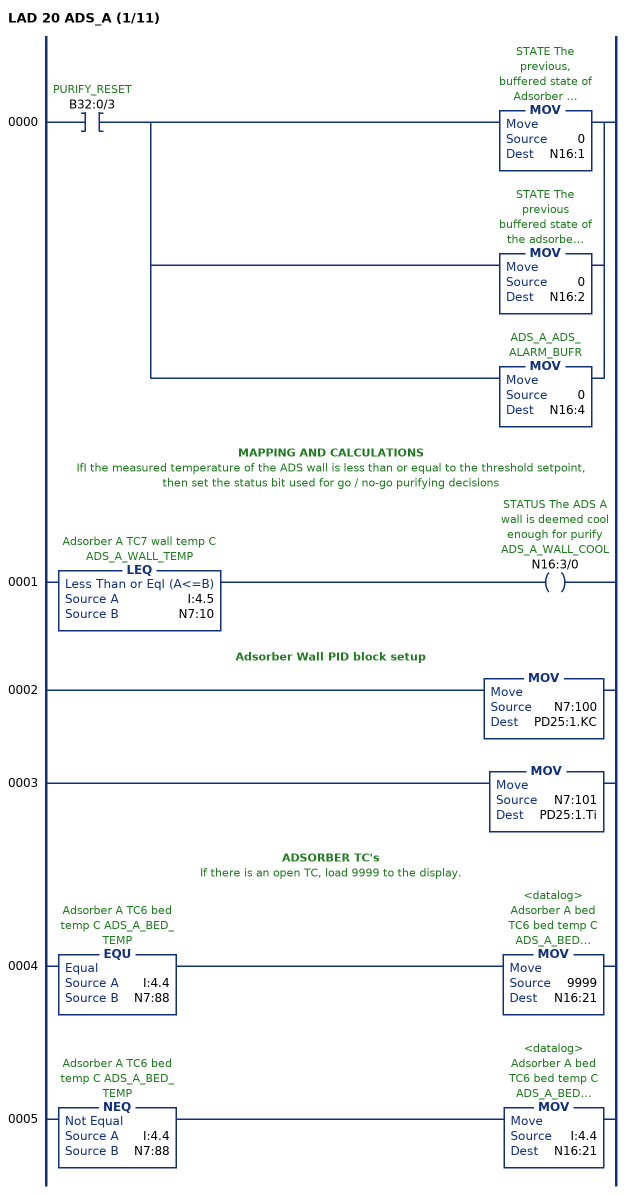
% Rung: 0 %
SOR XIC B32:0/3 BST MOV 0 N16:1 NXB MOV 0 N16:2 NXB MOV 0 N16:4 BND EOR
%   B32:0/3  PURIFY_RESET %
%   N16:1  ADS_A_STANDBY_BUFFER  "STATE The previous, buffered state of Adsorber A" %
%   N16:2  ADS_A_SYS_ALARM_BUFR  "STATE The previous buffered state of the adsorber when the alarm occured" %
%   N16:4  ADS_A_ADS_ALARM_BUFR %
% Rung: 1 %
% TITLE: MAPPING AND CALCULATIONS %
% IfI the measured temperature of the ADS wall is less than or equal to the threshold setpoint, then set the status bit used for go / no-go purifying decisions %
SOR LEQ I:4.5 N7:10 OTE N16:3/0 EOR
%   I:4.5  ADS_A_WALL_TEMP  "Adsorber A TC7 wall temp C" %
%   N7:10  ADS_WALL_TEMP_COOL  "CONFIG The temp at which the adsorber wall is deemed to be cool enough to purify" %
%   N16:3/0  ADS_A_WALL_COOL  "STATUS The ADS A wall is deemed cool enough for purify" %
% Rung: 2 %
% TITLE: Adsorber Wall PID block setup %
SOR MOV N7:100 PD25:1.KC EOR
%   N7:100  BLANKET_P  "CONFIG Blanket Proportional Gain New" %
% Rung: 3 %
SOR MOV N7:101 PD25:1.Ti EOR
%   N7:101  BLANKET_I  "CONFIG Blanket Integral Gain New" %
% Rung: 4 %
% TITLE: ADSORBER TC's %
% If there is an open TC, load 9999 to the display. %
SOR EQU I:4.4 N7:88 MOV 9999 N16:21 EOR
%   I:4.4  ADS_A_BED_TEMP  "Adsorber A TC6 bed temp C" %
%   N7:88  TC_OPEN_SP  "CONFIG The value read by an open TC input" %
%   N16:21  ADS_A_BED_TEMP_READ  "<datalog> Adsorber A bed TC6 bed temp C" %
% Rung: 5 %
SOR NEQ I:4.4 N7:88 MOV I:4.4 N16:21 EOR
%   I:4.4  ADS_A_BED_TEMP  "Adsorber A TC6 bed temp C" %
%   N7:88  TC_OPEN_SP  "CONFIG The value read by an open TC input" %
%   N16:21  ADS_A_BED_TEMP_READ  "<datalog> Adsorber A bed TC6 bed temp C" %

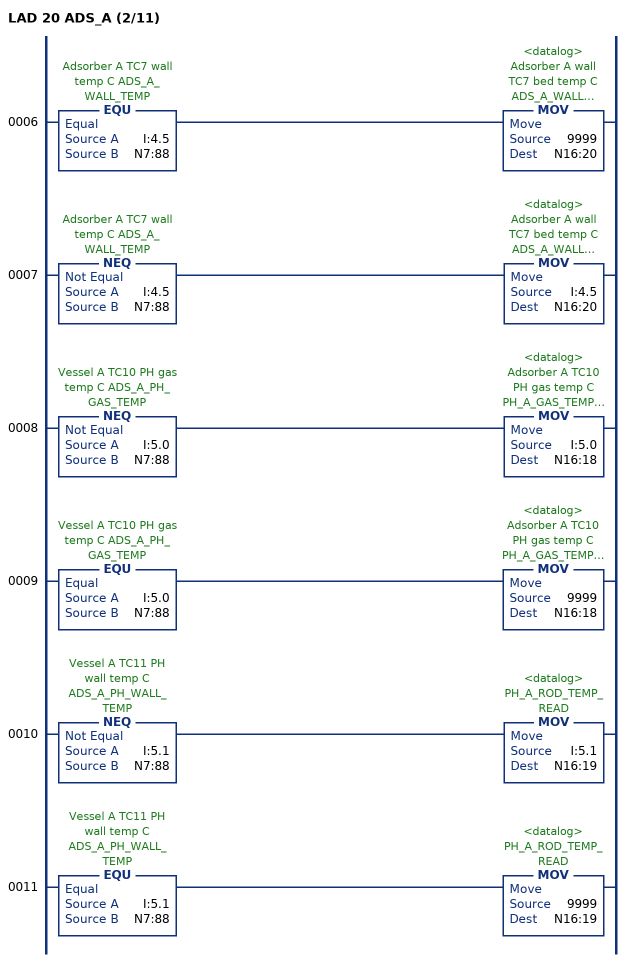
% Rung: 6 %
SOR EQU I:4.5 N7:88 MOV 9999 N16:20 EOR
%   I:4.5  ADS_A_WALL_TEMP  "Adsorber A TC7 wall temp C" %
%   N7:88  TC_OPEN_SP  "CONFIG The value read by an open TC input" %
%   N16:20  ADS_A_WALL_TEMP_READ  "<datalog> Adsorber A wall TC7 bed temp C" %
% Rung: 7 %
SOR NEQ I:4.5 N7:88 MOV I:4.5 N16:20 EOR
%   I:4.5  ADS_A_WALL_TEMP  "Adsorber A TC7 wall temp C" %
%   N7:88  TC_OPEN_SP  "CONFIG The value read by an open TC input" %
%   N16:20  ADS_A_WALL_TEMP_READ  "<datalog> Adsorber A wall TC7 bed temp C" %
% Rung: 8 %
SOR NEQ I:5.0 N7:88 MOV I:5.0 N16:18 EOR
%   I:5.0  ADS_A_PH_GAS_TEMP  "Vessel A TC10 PH gas temp C" %
%   N7:88  TC_OPEN_SP  "CONFIG The value read by an open TC input" %
%   N16:18  PH_A_GAS_TEMP_READ  "<datalog> Adsorber A TC10 PH gas temp C" %
% Rung: 9 %
SOR EQU I:5.0 N7:88 MOV 9999 N16:18 EOR
%   I:5.0  ADS_A_PH_GAS_TEMP  "Vessel A TC10 PH gas temp C" %
%   N7:88  TC_OPEN_SP  "CONFIG The value read by an open TC input" %
%   N16:18  PH_A_GAS_TEMP_READ  "<datalog> Adsorber A TC10 PH gas temp C" %
% Rung: 10 %
SOR NEQ I:5.1 N7:88 MOV I:5.1 N16:19 EOR
%   I:5.1  ADS_A_PH_WALL_TEMP  "Vessel A TC11 PH wall temp C" %
%   N7:88  TC_OPEN_SP  "CONFIG The value read by an open TC input" %
%   N16:19  PH_A_ROD_TEMP_READ  "<datalog>" %
% Rung: 11 %
SOR EQU I:5.1 N7:88 MOV 9999 N16:19 EOR
%   I:5.1  ADS_A_PH_WALL_TEMP  "Vessel A TC11 PH wall temp C" %
%   N7:88  TC_OPEN_SP  "CONFIG The value read by an open TC input" %
%   N16:19  PH_A_ROD_TEMP_READ  "<datalog>" %

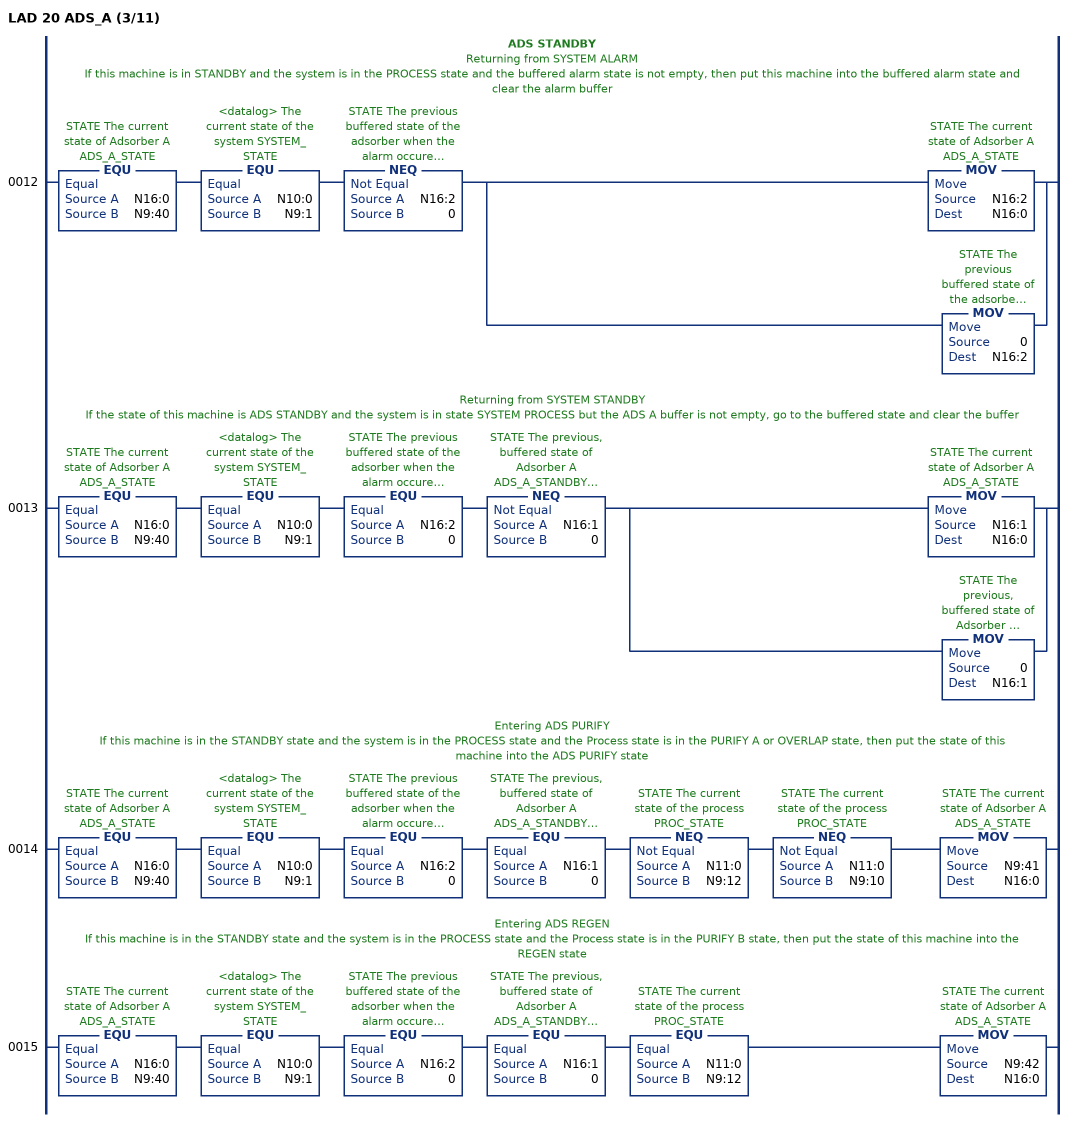
% Rung: 12 %
% TITLE: ADS STANDBY %
% Returning from SYSTEM ALARM
% If this machine is in STANDBY and the system is in the PROCESS state and the buffered alarm state is not empty, then put this machine into the buffered alarm state and clear the alarm buffer %
SOR EQU N16:0 N9:40 EQU N10:0 N9:1 NEQ N16:2 0 BST MOV N16:2 N16:0 NXB MOV 0 N16:2 BND EOR
%   N16:0  ADS_A_STATE  "STATE The current state of Adsorber A" %
%   N9:40  ADS_STANDBY  "STATE ADS Standby" %
%   N10:0  SYSTEM_STATE  "<datalog> The current state of the system" %
%   N9:1  SYSTEM_PROCESS  "STATE System Process" %
%   N16:2  ADS_A_SYS_ALARM_BUFR  "STATE The previous buffered state of the adsorber when the alarm occured" %
% Rung: 13 %
% Returning from SYSTEM STANDBY
% If the state of this machine is ADS STANDBY and the system is in state SYSTEM PROCESS but the ADS A buffer is not empty, go to the buffered state and clear the buffer %
SOR EQU N16:0 N9:40 EQU N10:0 N9:1 EQU N16:2 0 NEQ N16:1 0 BST MOV N16:1 N16:0 NXB MOV 0 N16:1 BND EOR
%   N16:0  ADS_A_STATE  "STATE The current state of Adsorber A" %
%   N9:40  ADS_STANDBY  "STATE ADS Standby" %
%   N10:0  SYSTEM_STATE  "<datalog> The current state of the system" %
%   N9:1  SYSTEM_PROCESS  "STATE System Process" %
%   N16:2  ADS_A_SYS_ALARM_BUFR  "STATE The previous buffered state of the adsorber when the alarm occured" %
%   N16:1  ADS_A_STANDBY_BUFFER  "STATE The previous, buffered state of Adsorber A" %
% Rung: 14 %
% Entering ADS PURIFY
% If this machine is in the STANDBY state and the system is in the PROCESS state and the Process state is in the PURIFY A or OVERLAP state, then put the state of this machine into the ADS PURIFY state %
SOR EQU N16:0 N9:40 EQU N10:0 N9:1 EQU N16:2 0 EQU N16:1 0 NEQ N11:0 N9:12 NEQ N11:0 N9:10 MOV N9:41 N16:0 EOR
%   N16:0  ADS_A_STATE  "STATE The current state of Adsorber A" %
%   N9:40  ADS_STANDBY  "STATE ADS Standby" %
%   N10:0  SYSTEM_STATE  "<datalog> The current state of the system" %
%   N9:1  SYSTEM_PROCESS  "STATE System Process" %
%   N16:2  ADS_A_SYS_ALARM_BUFR  "STATE The previous buffered state of the adsorber when the alarm occured" %
%   N16:1  ADS_A_STANDBY_BUFFER  "STATE The previous, buffered state of Adsorber A" %
%   N11:0  PROC_STATE  "STATE The current state of the process" %
%   N9:12  PROC_REGEN_A  "STATE Process Purify B" %
%   N9:10  PROCESS_STANDBY %
%   N9:41  ADS_PURIFY  "STATE ADS Purify" %
% Rung: 15 %
% Entering ADS REGEN
% If this machine is in the STANDBY state and the system is in the PROCESS state and the Process state is in the PURIFY B state, then put the state of this machine into the REGEN state %
SOR EQU N16:0 N9:40 EQU N10:0 N9:1 EQU N16:2 0 EQU N16:1 0 EQU N11:0 N9:12 MOV N9:42 N16:0 EOR
%   N16:0  ADS_A_STATE  "STATE The current state of Adsorber A" %
%   N9:40  ADS_STANDBY  "STATE ADS Standby" %
%   N10:0  SYSTEM_STATE  "<datalog> The current state of the system" %
%   N9:1  SYSTEM_PROCESS  "STATE System Process" %
%   N16:2  ADS_A_SYS_ALARM_BUFR  "STATE The previous buffered state of the adsorber when the alarm occured" %
%   N16:1  ADS_A_STANDBY_BUFFER  "STATE The previous, buffered state of Adsorber A" %
%   N11:0  PROC_STATE  "STATE The current state of the process" %
%   N9:12  PROC_REGEN_A  "STATE Process Purify B" %
%   N9:42  ADS_REGEN  "STATE ADS Regen" %

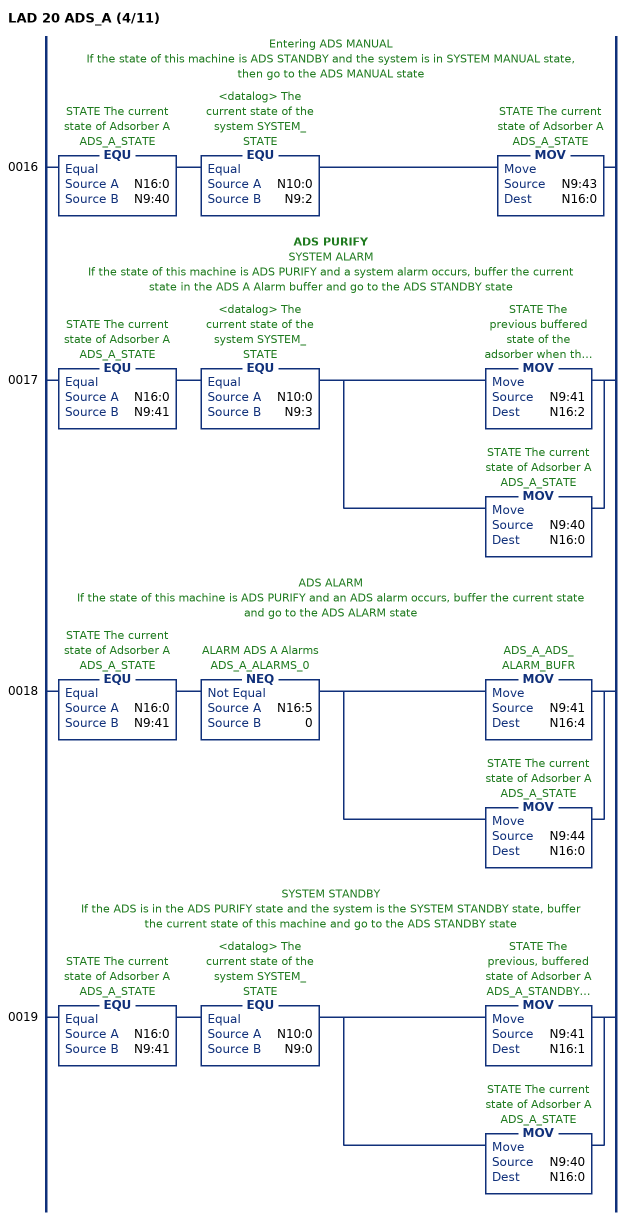
% Rung: 16 %
% Entering ADS MANUAL
% If the state of this machine is ADS STANDBY and the system is in SYSTEM MANUAL state, then go to the ADS MANUAL state %
SOR EQU N16:0 N9:40 EQU N10:0 N9:2 MOV N9:43 N16:0 EOR
%   N16:0  ADS_A_STATE  "STATE The current state of Adsorber A" %
%   N9:40  ADS_STANDBY  "STATE ADS Standby" %
%   N10:0  SYSTEM_STATE  "<datalog> The current state of the system" %
%   N9:2  SYSTEM_MANUAL  "STATE System Manual" %
%   N9:43  ADS_MANUAL  "STATE ADS Manual" %
% Rung: 17 %
% TITLE: ADS PURIFY %
% SYSTEM ALARM
% If the state of this machine is ADS PURIFY and a system alarm occurs, buffer the current state in the ADS A Alarm buffer and go to the ADS STANDBY state %
SOR EQU N16:0 N9:41 EQU N10:0 N9:3 BST MOV N9:41 N16:2 NXB MOV N9:40 N16:0 BND EOR
%   N16:0  ADS_A_STATE  "STATE The current state of Adsorber A" %
%   N9:41  ADS_PURIFY  "STATE ADS Purify" %
%   N10:0  SYSTEM_STATE  "<datalog> The current state of the system" %
%   N9:3  SYSTEM_ALARM  "STATE System Alarm" %
%   N16:2  ADS_A_SYS_ALARM_BUFR  "STATE The previous buffered state of the adsorber when the alarm occured" %
%   N9:40  ADS_STANDBY  "STATE ADS Standby" %
% Rung: 18 %
% ADS ALARM
% If the state of this machine is ADS PURIFY and an ADS alarm occurs, buffer the current state and go to the ADS ALARM state %
SOR EQU N16:0 N9:41 NEQ N16:5 0 BST MOV N9:41 N16:4 NXB MOV N9:44 N16:0 BND EOR
%   N16:0  ADS_A_STATE  "STATE The current state of Adsorber A" %
%   N9:41  ADS_PURIFY  "STATE ADS Purify" %
%   N16:5  ADS_A_ALARMS_0  "ALARM ADS A Alarms" %
%   N16:4  ADS_A_ADS_ALARM_BUFR %
%   N9:44  ADS_ALARM  "STATE ADS Alarm" %
% Rung: 19 %
% SYSTEM STANDBY
% If the ADS is in the ADS PURIFY state and the system is the SYSTEM STANDBY state, buffer the current state of this machine and go to the ADS STANDBY state %
SOR EQU N16:0 N9:41 EQU N10:0 N9:0 BST MOV N9:41 N16:1 NXB MOV N9:40 N16:0 BND EOR
%   N16:0  ADS_A_STATE  "STATE The current state of Adsorber A" %
%   N9:41  ADS_PURIFY  "STATE ADS Purify" %
%   N10:0  SYSTEM_STATE  "<datalog> The current state of the system" %
%   N9:0  SYSTEM_STANDBY  "STATE System Standby" %
%   N16:1  ADS_A_STANDBY_BUFFER  "STATE The previous, buffered state of Adsorber A" %
%   N9:40  ADS_STANDBY  "STATE ADS Standby" %

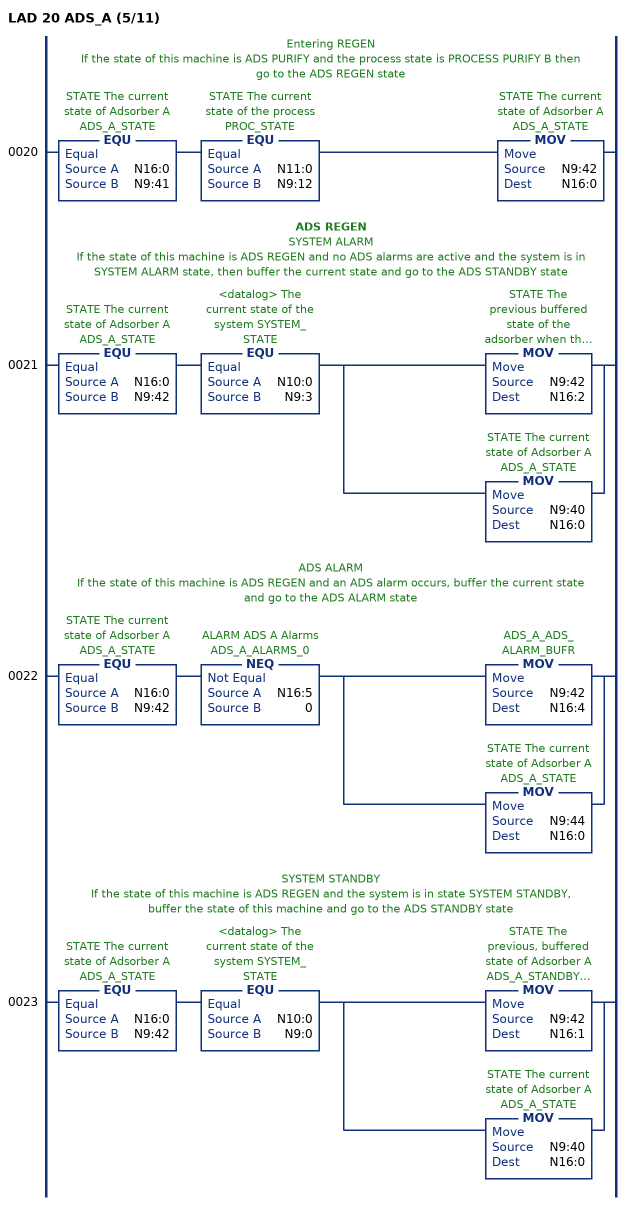
% Rung: 20 %
% Entering REGEN
% If the state of this machine is ADS PURIFY and the process state is PROCESS PURIFY B then go to the ADS REGEN state %
SOR EQU N16:0 N9:41 EQU N11:0 N9:12 MOV N9:42 N16:0 EOR
%   N16:0  ADS_A_STATE  "STATE The current state of Adsorber A" %
%   N9:41  ADS_PURIFY  "STATE ADS Purify" %
%   N11:0  PROC_STATE  "STATE The current state of the process" %
%   N9:12  PROC_REGEN_A  "STATE Process Purify B" %
%   N9:42  ADS_REGEN  "STATE ADS Regen" %
% Rung: 21 %
% TITLE: ADS REGEN %
% SYSTEM ALARM
% If the state of this machine is ADS REGEN and no ADS alarms are active and the system is in SYSTEM ALARM state, then buffer the current state and go to the ADS STANDBY state %
SOR EQU N16:0 N9:42 EQU N10:0 N9:3 BST MOV N9:42 N16:2 NXB MOV N9:40 N16:0 BND EOR
%   N16:0  ADS_A_STATE  "STATE The current state of Adsorber A" %
%   N9:42  ADS_REGEN  "STATE ADS Regen" %
%   N10:0  SYSTEM_STATE  "<datalog> The current state of the system" %
%   N9:3  SYSTEM_ALARM  "STATE System Alarm" %
%   N16:2  ADS_A_SYS_ALARM_BUFR  "STATE The previous buffered state of the adsorber when the alarm occured" %
%   N9:40  ADS_STANDBY  "STATE ADS Standby" %
% Rung: 22 %
% ADS ALARM
% If the state of this machine is ADS REGEN and an ADS alarm occurs, buffer the current state and go to the ADS ALARM state %
SOR EQU N16:0 N9:42 NEQ N16:5 0 BST MOV N9:42 N16:4 NXB MOV N9:44 N16:0 BND EOR
%   N16:0  ADS_A_STATE  "STATE The current state of Adsorber A" %
%   N9:42  ADS_REGEN  "STATE ADS Regen" %
%   N16:5  ADS_A_ALARMS_0  "ALARM ADS A Alarms" %
%   N16:4  ADS_A_ADS_ALARM_BUFR %
%   N9:44  ADS_ALARM  "STATE ADS Alarm" %
% Rung: 23 %
% SYSTEM STANDBY
% If the state of this machine is ADS REGEN and the system is in state SYSTEM STANDBY, buffer the state of this machine and go to the ADS STANDBY state %
SOR EQU N16:0 N9:42 EQU N10:0 N9:0 BST MOV N9:42 N16:1 NXB MOV N9:40 N16:0 BND EOR
%   N16:0  ADS_A_STATE  "STATE The current state of Adsorber A" %
%   N9:42  ADS_REGEN  "STATE ADS Regen" %
%   N10:0  SYSTEM_STATE  "<datalog> The current state of the system" %
%   N9:0  SYSTEM_STANDBY  "STATE System Standby" %
%   N16:1  ADS_A_STANDBY_BUFFER  "STATE The previous, buffered state of Adsorber A" %
%   N9:40  ADS_STANDBY  "STATE ADS Standby" %

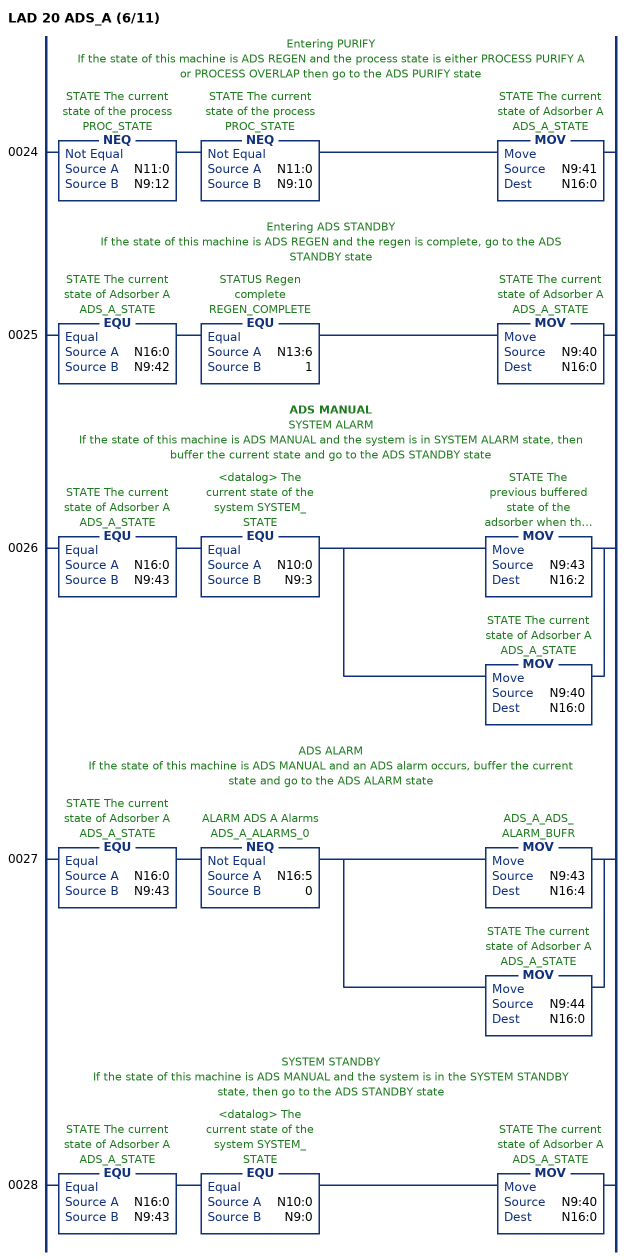
% Rung: 24 %
% Entering PURIFY
% If the state of this machine is ADS REGEN and the process state is either PROCESS PURIFY A or PROCESS OVERLAP then go to the ADS PURIFY state %
SOR NEQ N11:0 N9:12 NEQ N11:0 N9:10 MOV N9:41 N16:0 EOR
%   N11:0  PROC_STATE  "STATE The current state of the process" %
%   N9:12  PROC_REGEN_A  "STATE Process Purify B" %
%   N9:10  PROCESS_STANDBY %
%   N9:41  ADS_PURIFY  "STATE ADS Purify" %
%   N16:0  ADS_A_STATE  "STATE The current state of Adsorber A" %
% Rung: 25 %
% Entering ADS STANDBY
% If the state of this machine is ADS REGEN and the regen is complete, go to the ADS STANDBY state %
SOR EQU N16:0 N9:42 EQU N13:6 1 MOV N9:40 N16:0 EOR
%   N16:0  ADS_A_STATE  "STATE The current state of Adsorber A" %
%   N9:42  ADS_REGEN  "STATE ADS Regen" %
%   N13:6  REGEN_COMPLETE  "STATUS Regen complete" %
%   N9:40  ADS_STANDBY  "STATE ADS Standby" %
% Rung: 26 %
% TITLE: ADS MANUAL %
% SYSTEM ALARM
% If the state of this machine is ADS MANUAL and the system is in SYSTEM ALARM state, then buffer the current state and go to the ADS STANDBY state %
SOR EQU N16:0 N9:43 EQU N10:0 N9:3 BST MOV N9:43 N16:2 NXB MOV N9:40 N16:0 BND EOR
%   N16:0  ADS_A_STATE  "STATE The current state of Adsorber A" %
%   N9:43  ADS_MANUAL  "STATE ADS Manual" %
%   N10:0  SYSTEM_STATE  "<datalog> The current state of the system" %
%   N9:3  SYSTEM_ALARM  "STATE System Alarm" %
%   N16:2  ADS_A_SYS_ALARM_BUFR  "STATE The previous buffered state of the adsorber when the alarm occured" %
%   N9:40  ADS_STANDBY  "STATE ADS Standby" %
% Rung: 27 %
% ADS ALARM
% If the state of this machine is ADS MANUAL and an ADS alarm occurs, buffer the current state and go to the ADS ALARM state %
SOR EQU N16:0 N9:43 NEQ N16:5 0 BST MOV N9:43 N16:4 NXB MOV N9:44 N16:0 BND EOR
%   N16:0  ADS_A_STATE  "STATE The current state of Adsorber A" %
%   N9:43  ADS_MANUAL  "STATE ADS Manual" %
%   N16:5  ADS_A_ALARMS_0  "ALARM ADS A Alarms" %
%   N16:4  ADS_A_ADS_ALARM_BUFR %
%   N9:44  ADS_ALARM  "STATE ADS Alarm" %
% Rung: 28 %
% SYSTEM STANDBY
% If the state of this machine is ADS MANUAL and the system is in the SYSTEM STANDBY state, then go to the ADS STANDBY state %
SOR EQU N16:0 N9:43 EQU N10:0 N9:0 MOV N9:40 N16:0 EOR
%   N16:0  ADS_A_STATE  "STATE The current state of Adsorber A" %
%   N9:43  ADS_MANUAL  "STATE ADS Manual" %
%   N10:0  SYSTEM_STATE  "<datalog> The current state of the system" %
%   N9:0  SYSTEM_STANDBY  "STATE System Standby" %
%   N9:40  ADS_STANDBY  "STATE ADS Standby" %

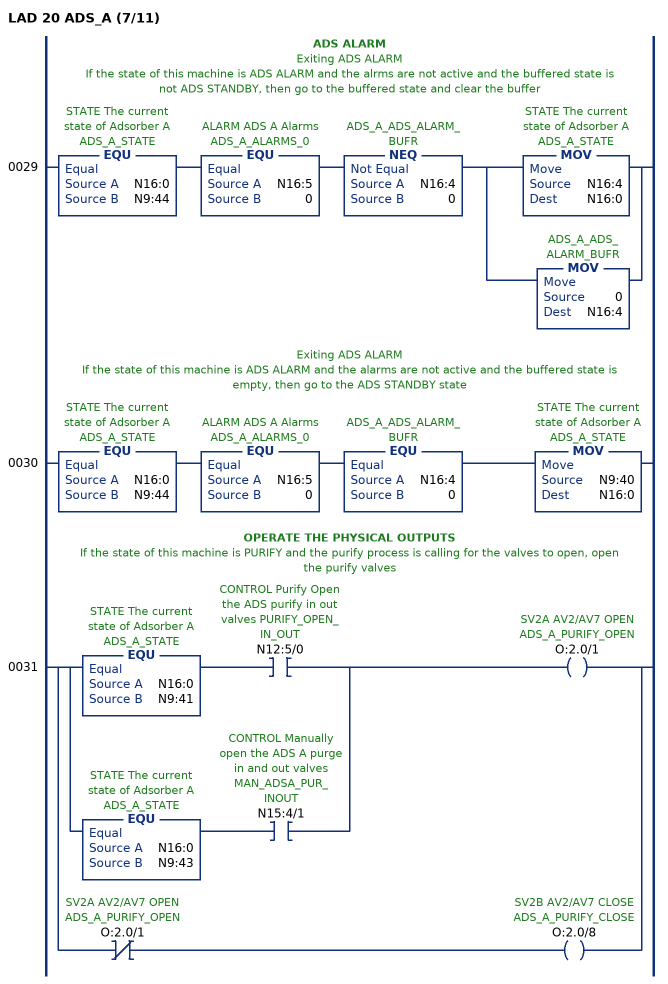
% Rung: 29 %
% TITLE: ADS ALARM %
% Exiting ADS ALARM
% If the state of this machine is ADS ALARM and the alrms are not active and the buffered state is not ADS STANDBY, then go to the buffered state and clear the buffer %
SOR EQU N16:0 N9:44 EQU N16:5 0 NEQ N16:4 0 BST MOV N16:4 N16:0 NXB MOV 0 N16:4 BND EOR
%   N16:0  ADS_A_STATE  "STATE The current state of Adsorber A" %
%   N9:44  ADS_ALARM  "STATE ADS Alarm" %
%   N16:5  ADS_A_ALARMS_0  "ALARM ADS A Alarms" %
%   N16:4  ADS_A_ADS_ALARM_BUFR %
% Rung: 30 %
% Exiting ADS ALARM
% If the state of this machine is ADS ALARM and the alarms are not active and the buffered state is empty, then go to the ADS STANDBY state %
SOR EQU N16:0 N9:44 EQU N16:5 0 EQU N16:4 0 MOV N9:40 N16:0 EOR
%   N16:0  ADS_A_STATE  "STATE The current state of Adsorber A" %
%   N9:44  ADS_ALARM  "STATE ADS Alarm" %
%   N16:5  ADS_A_ALARMS_0  "ALARM ADS A Alarms" %
%   N16:4  ADS_A_ADS_ALARM_BUFR %
%   N9:40  ADS_STANDBY  "STATE ADS Standby" %
% Rung: 31 %
% TITLE: OPERATE THE PHYSICAL OUTPUTS %
% If the state of this machine is PURIFY and the purify process is calling for the valves to open, open the purify valves %
SOR BST BST EQU N16:0 N9:41 XIC N12:5/0 NXB EQU N16:0 N9:43 XIC N15:4/1 BND OTE O:2.0/1 NXB XIO O:2.0/1 OTE O:2.0/8 BND EOR
%   N16:0  ADS_A_STATE  "STATE The current state of Adsorber A" %
%   N9:41  ADS_PURIFY  "STATE ADS Purify" %
%   N12:5/0  PURIFY_OPEN_IN_OUT  "CONTROL Purify Open the ADS purify in out valves" %
%   N9:43  ADS_MANUAL  "STATE ADS Manual" %
%   N15:4/1  MAN_ADSA_PUR_INOUT  "CONTROL Manually open the ADS A purge in and out valves" %
%   O:2.0/1  ADS_A_PURIFY_OPEN  "SV2A AV2/AV7 OPEN" %
%   O:2.0/8  ADS_A_PURIFY_CLOSE  "SV2B AV2/AV7 CLOSE" %

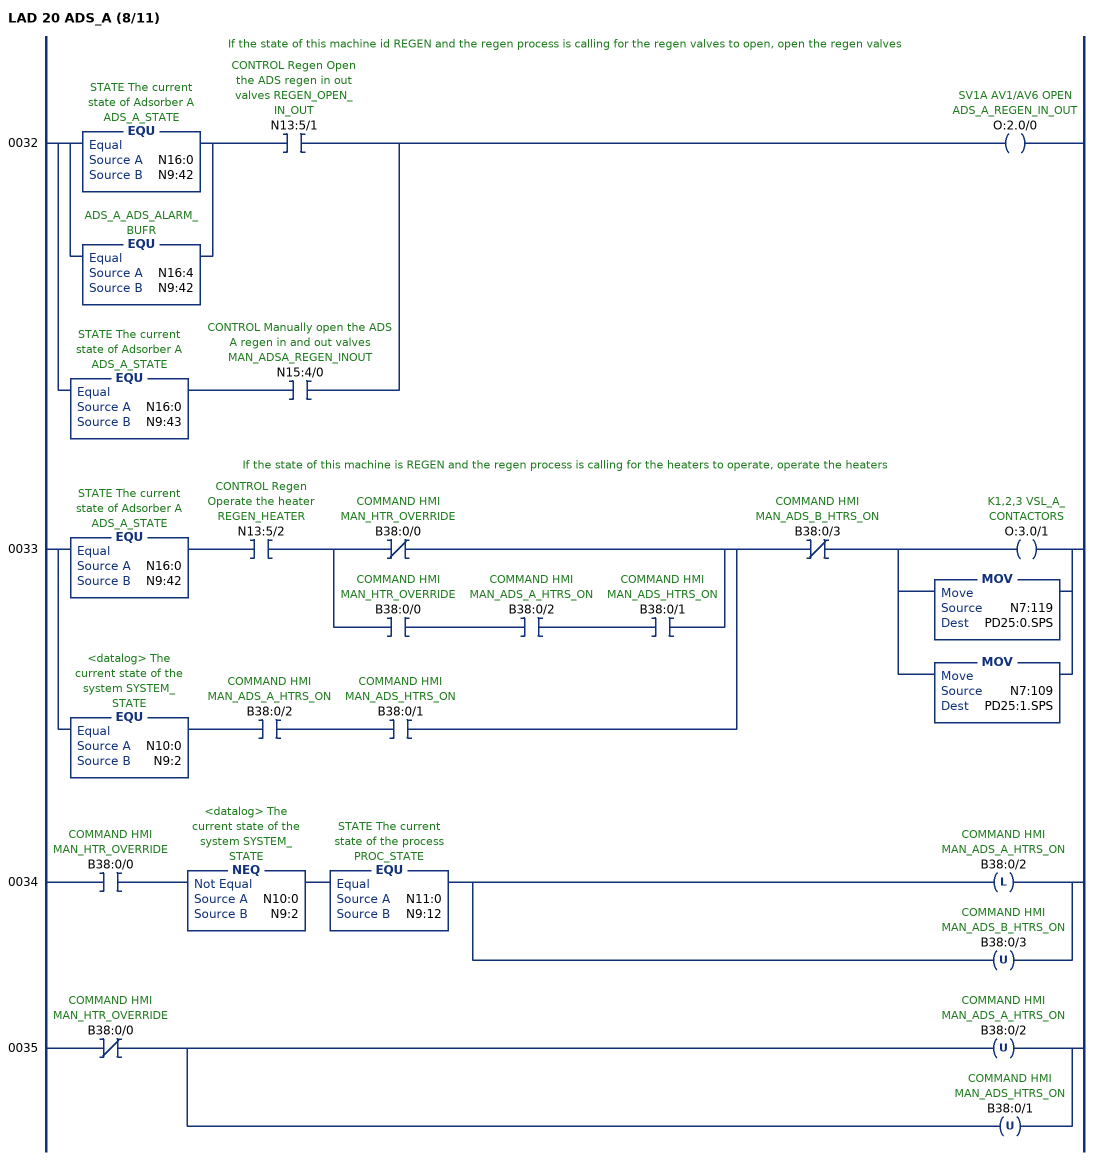
% Rung: 32 %
% If the state of this machine id REGEN and the regen process is calling for the regen valves to open, open the regen valves %
SOR BST BST EQU N16:0 N9:42 NXB EQU N16:4 N9:42 BND XIC N13:5/1 NXB EQU N16:0 N9:43 XIC N15:4/0 BND OTE O:2.0/0 EOR
%   N16:0  ADS_A_STATE  "STATE The current state of Adsorber A" %
%   N9:42  ADS_REGEN  "STATE ADS Regen" %
%   N16:4  ADS_A_ADS_ALARM_BUFR %
%   N13:5/1  REGEN_OPEN_IN_OUT  "CONTROL Regen Open the ADS regen in out valves" %
%   N9:43  ADS_MANUAL  "STATE ADS Manual" %
%   N15:4/0  MAN_ADSA_REGEN_INOUT  "CONTROL Manually open the ADS A regen in and out valves" %
%   O:2.0/0  ADS_A_REGEN_IN_OUT  "SV1A AV1/AV6 OPEN" %
% Rung: 33 %
% If the state of this machine is REGEN and the regen process is calling for the heaters to operate, operate the heaters %
SOR BST EQU N16:0 N9:42 XIC N13:5/2 BST XIO B38:0/0 NXB XIC B38:0/0 XIC B38:0/2 XIC B38:0/1 BND NXB EQU N10:0 N9:2 XIC B38:0/2 XIC B38:0/1 BND XIO B38:0/3 BST OTE O:3.0/1 NXB MOV N7:119 PD25:0.SPS NXB MOV N7:109 PD25:1.SPS BND EOR
%   N16:0  ADS_A_STATE  "STATE The current state of Adsorber A" %
%   N9:42  ADS_REGEN  "STATE ADS Regen" %
%   N13:5/2  REGEN_HEATER  "CONTROL Regen Operate the heater" %
%   B38:0/0  MAN_HTR_OVERRIDE  "COMMAND HMI" %
%   B38:0/2  MAN_ADS_A_HTRS_ON  "COMMAND HMI" %
%   B38:0/1  MAN_ADS_HTRS_ON  "COMMAND HMI" %
%   N10:0  SYSTEM_STATE  "<datalog> The current state of the system" %
%   N9:2  SYSTEM_MANUAL  "STATE System Manual" %
%   B38:0/3  MAN_ADS_B_HTRS_ON  "COMMAND HMI" %
%   O:3.0/1  VSL_A_CONTACTORS  "K1,2,3" %
%   N7:119  PREHEATER_SP  "<datalog> CONTROL Preheater PID Setpoint" %
%   N7:109  BLANKET_SP  "CONTROL Blanket PID Setpoint" %
% Rung: 34 %
SOR XIC B38:0/0 NEQ N10:0 N9:2 EQU N11:0 N9:12 BST OTL B38:0/2 NXB OTU B38:0/3 BND EOR
%   B38:0/0  MAN_HTR_OVERRIDE  "COMMAND HMI" %
%   N10:0  SYSTEM_STATE  "<datalog> The current state of the system" %
%   N9:2  SYSTEM_MANUAL  "STATE System Manual" %
%   N11:0  PROC_STATE  "STATE The current state of the process" %
%   N9:12  PROC_REGEN_A  "STATE Process Purify B" %
%   B38:0/2  MAN_ADS_A_HTRS_ON  "COMMAND HMI" %
%   B38:0/3  MAN_ADS_B_HTRS_ON  "COMMAND HMI" %
% Rung: 35 %
SOR XIO B38:0/0 BST OTU B38:0/2 NXB OTU B38:0/1 BND EOR
%   B38:0/0  MAN_HTR_OVERRIDE  "COMMAND HMI" %
%   B38:0/2  MAN_ADS_A_HTRS_ON  "COMMAND HMI" %
%   B38:0/1  MAN_ADS_HTRS_ON  "COMMAND HMI" %

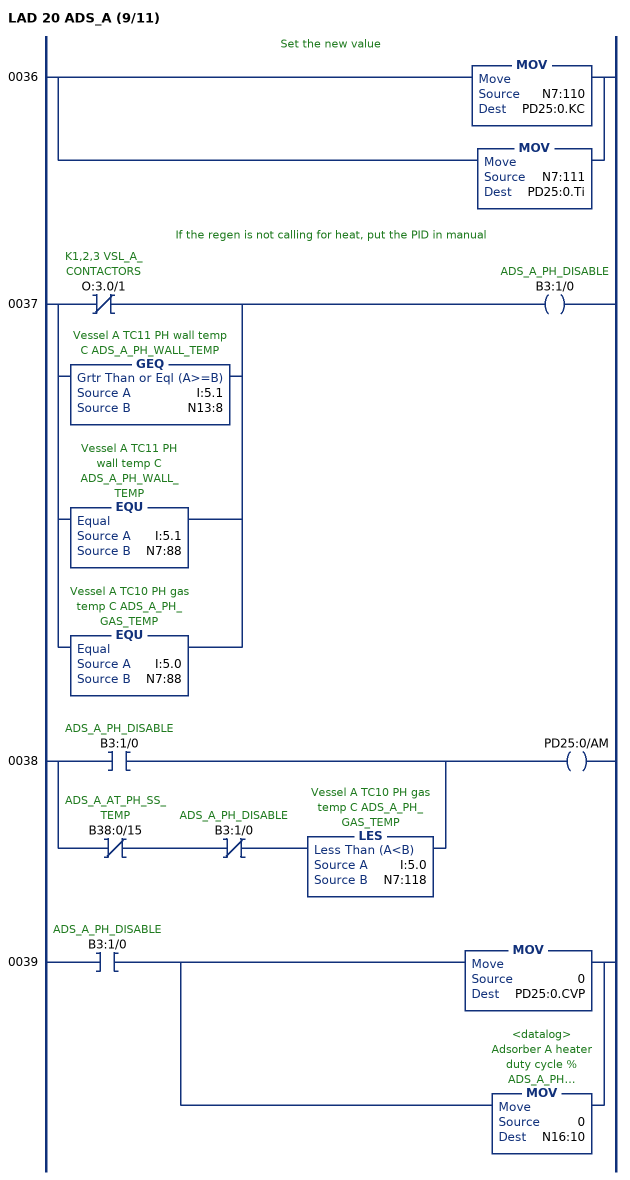
% Rung: 36 %
% Set the new value %
SOR BST MOV N7:110 PD25:0.KC NXB MOV N7:111 PD25:0.Ti BND EOR
%   N7:110  PREHEATER_P  "<datalog> CONFIG Preheater Proportional Gain New" %
%   N7:111  PREHEATER_I  "<datalog> CONFIG Preheater Integral Gain New" %
% Rung: 37 %
% If the regen is not calling for heat, put the PID in manual %
SOR BST XIO O:3.0/1 NXB GEQ I:5.1 N13:8 NXB EQU I:5.1 N7:88 NXB EQU I:5.0 N7:88 BND OTE B3:1/0 EOR
%   O:3.0/1  VSL_A_CONTACTORS  "K1,2,3" %
%   I:5.1  ADS_A_PH_WALL_TEMP  "Vessel A TC11 PH wall temp C" %
%   N13:8  PH_ROD_LIMIT %
%   N7:88  TC_OPEN_SP  "CONFIG The value read by an open TC input" %
%   I:5.0  ADS_A_PH_GAS_TEMP  "Vessel A TC10 PH gas temp C" %
%   B3:1/0  ADS_A_PH_DISABLE %
% Rung: 38 %
SOR BST XIC B3:1/0 NXB XIO B38:0/15 XIO B3:1/0 LES I:5.0 N7:118 BND OTE PD25:0/AM EOR
%   B3:1/0  ADS_A_PH_DISABLE %
%   B38:0/15  ADS_A_AT_PH_SS_TEMP %
%   I:5.0  ADS_A_PH_GAS_TEMP  "Vessel A TC10 PH gas temp C" %
%   N7:118  PH_SS_TEMP_SP %
% Rung: 39 %
SOR XIC B3:1/0 BST MOV 0 PD25:0.CVP NXB MOV 0 N16:10 BND EOR
%   B3:1/0  ADS_A_PH_DISABLE %
%   N16:10  ADS_A_PH_OUTPUT  "<datalog> Adsorber A heater duty cycle %" %

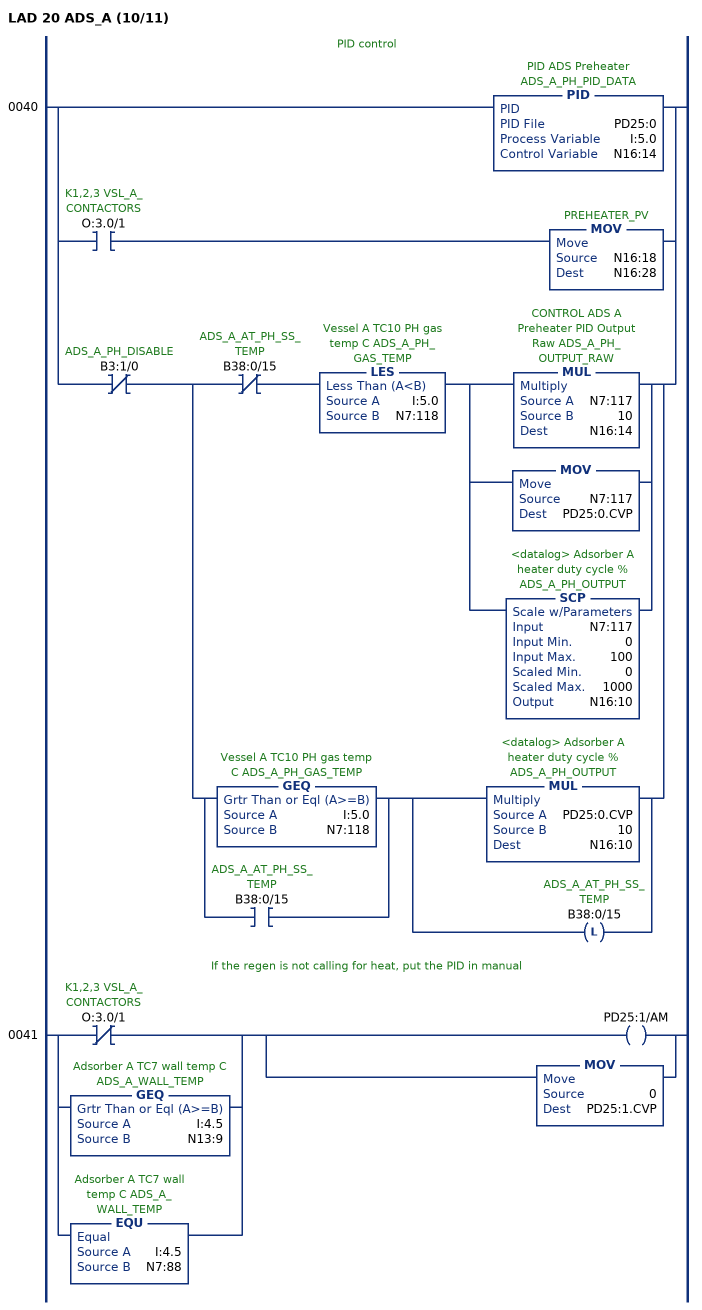
% Rung: 40 %
% PID control %
SOR BST PID PD25:0 I:5.0 N16:14 NXB XIC O:3.0/1 MOV N16:18 N16:28 NXB XIO B3:1/0 BST XIO B38:0/15 LES I:5.0 N7:118 BST MUL N7:117 10 N16:14 NXB MOV N7:117 PD25:0.CVP NXB SCP N7:117 0 100 0 1000 N16:10 BND NXB BST GEQ I:5.0 N7:118 NXB XIC B38:0/15 BND BST MUL PD25:0.CVP 10 N16:10 NXB OTL B38:0/15 BND BND BND EOR
%   PD25:0  ADS_A_PH_PID_DATA  "PID ADS Preheater" %
%   I:5.0  ADS_A_PH_GAS_TEMP  "Vessel A TC10 PH gas temp C" %
%   N16:14  ADS_A_PH_OUTPUT_RAW  "CONTROL ADS A Preheater PID Output Raw" %
%   O:3.0/1  VSL_A_CONTACTORS  "K1,2,3" %
%   N16:18  PH_A_GAS_TEMP_READ  "<datalog> Adsorber A TC10 PH gas temp C" %
%   N16:28  PREHEATER_PV %
%   B3:1/0  ADS_A_PH_DISABLE %
%   B38:0/15  ADS_A_AT_PH_SS_TEMP %
%   N7:118  PH_SS_TEMP_SP %
%   N7:117  PH_SS_OUTPUT %
%   N16:10  ADS_A_PH_OUTPUT  "<datalog> Adsorber A heater duty cycle %" %
% Rung: 41 %
% If the regen is not calling for heat, put the PID in manual %
SOR BST XIO O:3.0/1 NXB GEQ I:4.5 N13:9 NXB EQU I:4.5 N7:88 BND BST OTE PD25:1/AM NXB MOV 0 PD25:1.CVP BND EOR
%   O:3.0/1  VSL_A_CONTACTORS  "K1,2,3" %
%   I:4.5  ADS_A_WALL_TEMP  "Adsorber A TC7 wall temp C" %
%   N13:9  BLANKET_LIMIT %
%   N7:88  TC_OPEN_SP  "CONFIG The value read by an open TC input" %

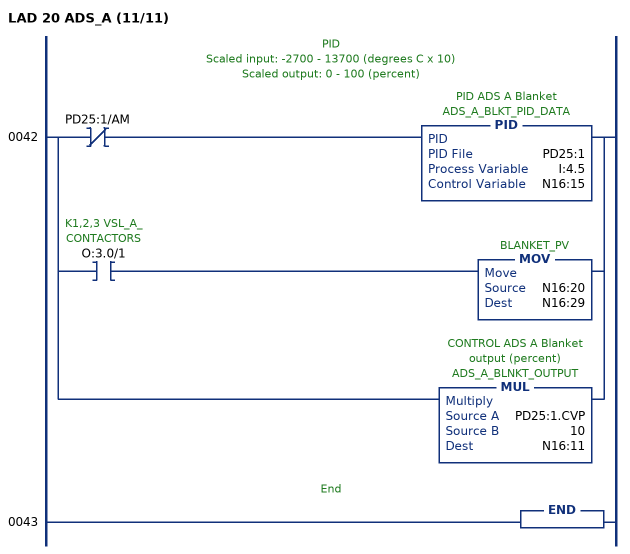
% Rung: 42 %
% PID
% Scaled input: -2700 - 13700 (degrees C x 10)
% Scaled output: 0 - 100 (percent) %
SOR BST XIO PD25:1/AM PID PD25:1 I:4.5 N16:15 NXB XIC O:3.0/1 MOV N16:20 N16:29 NXB MUL PD25:1.CVP 10 N16:11 BND EOR
%   PD25:1  ADS_A_BLKT_PID_DATA  "PID ADS A Blanket" %
%   I:4.5  ADS_A_WALL_TEMP  "Adsorber A TC7 wall temp C" %
%   N16:15  ADS_A_BLKT_OUTPT_RAW  "CONTROL ADS A Blanket PID Output Raw" %
%   O:3.0/1  VSL_A_CONTACTORS  "K1,2,3" %
%   N16:20  ADS_A_WALL_TEMP_READ  "<datalog> Adsorber A wall TC7 bed temp C" %
%   N16:29  BLANKET_PV %
%   N16:11  ADS_A_BLNKT_OUTPUT  "CONTROL ADS A Blanket output (percent)" %
% Rung: 43 %
% End %
SOR END EOR

LADDER 21 "ADS_A_FLT"    % Controls the Adsorber A faults %
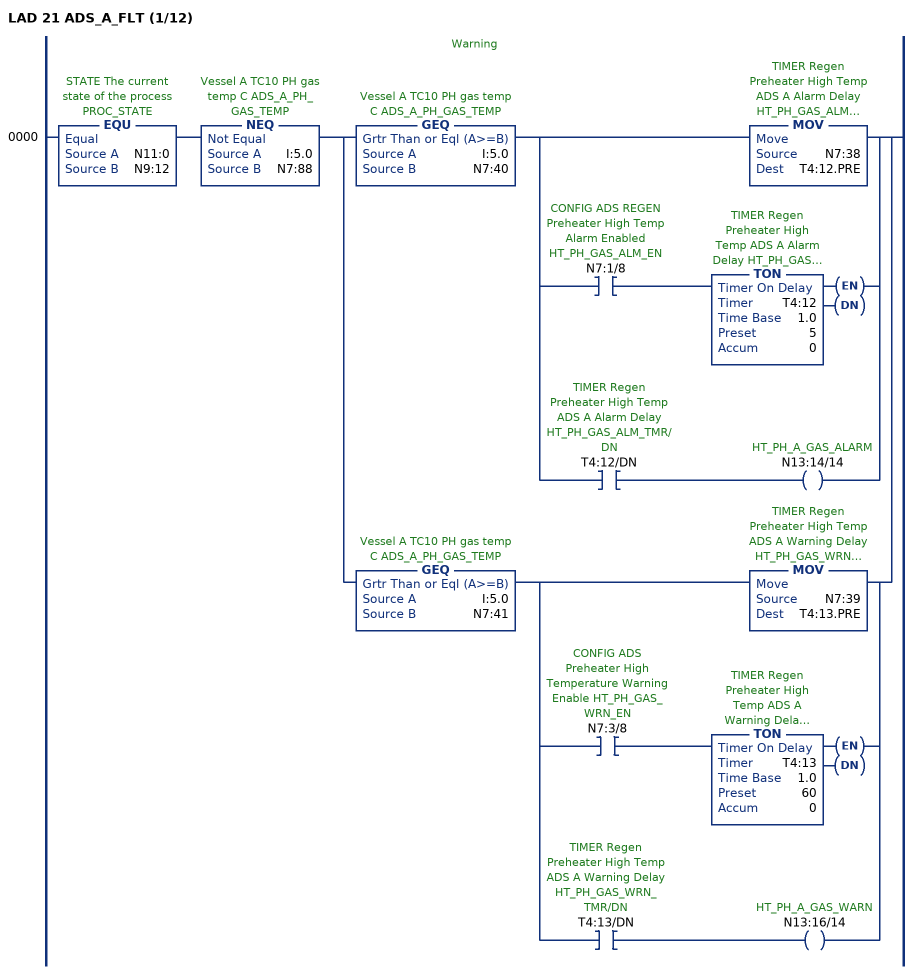
% Rung: 0 %
% Warning %
SOR EQU N11:0 N9:12 NEQ I:5.0 N7:88 BST GEQ I:5.0 N7:40 BST MOV N7:38 T4:12.PRE NXB XIC N7:1/8 TON T4:12 1.0 5 0 NXB XIC T4:12/DN OTE N13:14/14 BND NXB GEQ I:5.0 N7:41 BST MOV N7:39 T4:13.PRE NXB XIC N7:3/8 TON T4:13 1.0 60 0 NXB XIC T4:13/DN OTE N13:16/14 BND BND EOR
%   N11:0  PROC_STATE  "STATE The current state of the process" %
%   N9:12  PROC_REGEN_A  "STATE Process Purify B" %
%   I:5.0  ADS_A_PH_GAS_TEMP  "Vessel A TC10 PH gas temp C" %
%   N7:88  TC_OPEN_SP  "CONFIG The value read by an open TC input" %
%   N7:40  HT_PH_GAS_ALM_SP  "CONFIG ADS Preheater High Temperature Alarm Temperature" %
%   N7:38  HT_PH_GAS_ALM_DLY  "CONFIG ADS Preheater High Temperature Alarm Delay" %
%   T4:12  HT_PH_GAS_ALM_TMR  "TIMER Regen Preheater High Temp ADS A Alarm Delay" %
%   N7:1/8  HT_PH_GAS_ALM_EN  "CONFIG ADS REGEN Preheater High Temp Alarm Enabled" %
%   N13:14/14  HT_PH_A_GAS_ALARM %
%   N7:41  HT_PH_GAS_WRN_SP  "CONFIG ADS Preheater High Temperature Warning Temperature" %
%   N7:39  HT_PH_GAS_WRN_DLY  "CONFIG ADS Preheater High Temperature Warning Delay" %
%   T4:13  HT_PH_GAS_WRN_TMR  "TIMER Regen Preheater High Temp ADS A Warning Delay" %
%   N7:3/8  HT_PH_GAS_WRN_EN  "CONFIG ADS Preheater High Temperature Warning Enable" %
%   N13:16/14  HT_PH_A_GAS_WARN %

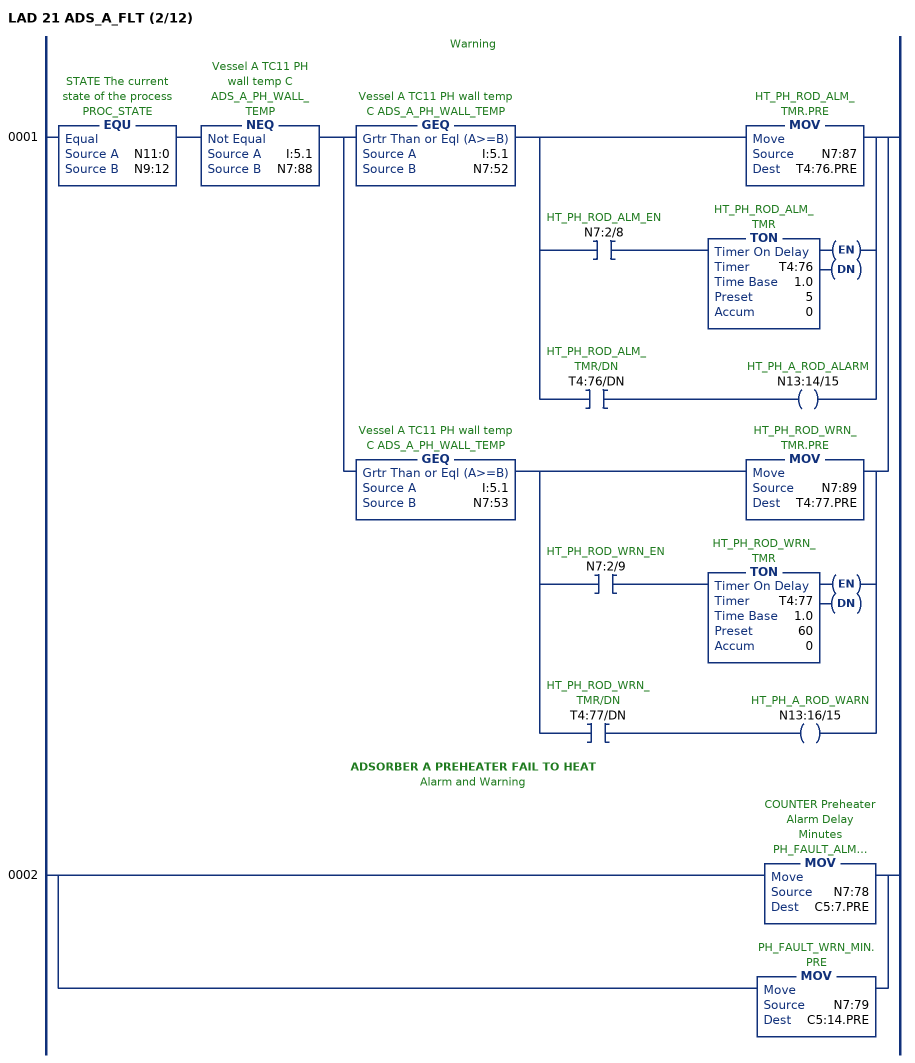
% Rung: 1 %
% Warning %
SOR EQU N11:0 N9:12 NEQ I:5.1 N7:88 BST GEQ I:5.1 N7:52 BST MOV N7:87 T4:76.PRE NXB XIC N7:2/8 TON T4:76 1.0 5 0 NXB XIC T4:76/DN OTE N13:14/15 BND NXB GEQ I:5.1 N7:53 BST MOV N7:89 T4:77.PRE NXB XIC N7:2/9 TON T4:77 1.0 60 0 NXB XIC T4:77/DN OTE N13:16/15 BND BND EOR
%   N11:0  PROC_STATE  "STATE The current state of the process" %
%   N9:12  PROC_REGEN_A  "STATE Process Purify B" %
%   I:5.1  ADS_A_PH_WALL_TEMP  "Vessel A TC11 PH wall temp C" %
%   N7:88  TC_OPEN_SP  "CONFIG The value read by an open TC input" %
%   N7:52  HT_PH_ROD_ALM_SP %
%   N7:87  HT_PH_ROD_ALM_DLY %
%   T4:76  HT_PH_ROD_ALM_TMR %
%   N7:2/8  HT_PH_ROD_ALM_EN %
%   N13:14/15  HT_PH_A_ROD_ALARM %
%   N7:53  HT_PH_ROD_WRN_SP %
%   N7:89  HT_PH_ROD_WRN_DLY %
%   T4:77  HT_PH_ROD_WRN_TMR %
%   N7:2/9  HT_PH_ROD_WRN_EN %
%   N13:16/15  HT_PH_A_ROD_WARN %
% Rung: 2 %
% TITLE: ADSORBER A PREHEATER FAIL TO HEAT %
% Alarm and Warning %
SOR BST MOV N7:78 C5:7.PRE NXB MOV N7:79 C5:14.PRE BND EOR
%   N7:78  PH_FAULT_ALM_DLY %
%   C5:7  PH_FAULT_ALM_MIN  "COUNTER Preheater Alarm Delay Minutes" %
%   N7:79  PH_FAULT_WRN_DLY %
%   C5:14  PH_FAULT_WRN_MIN %

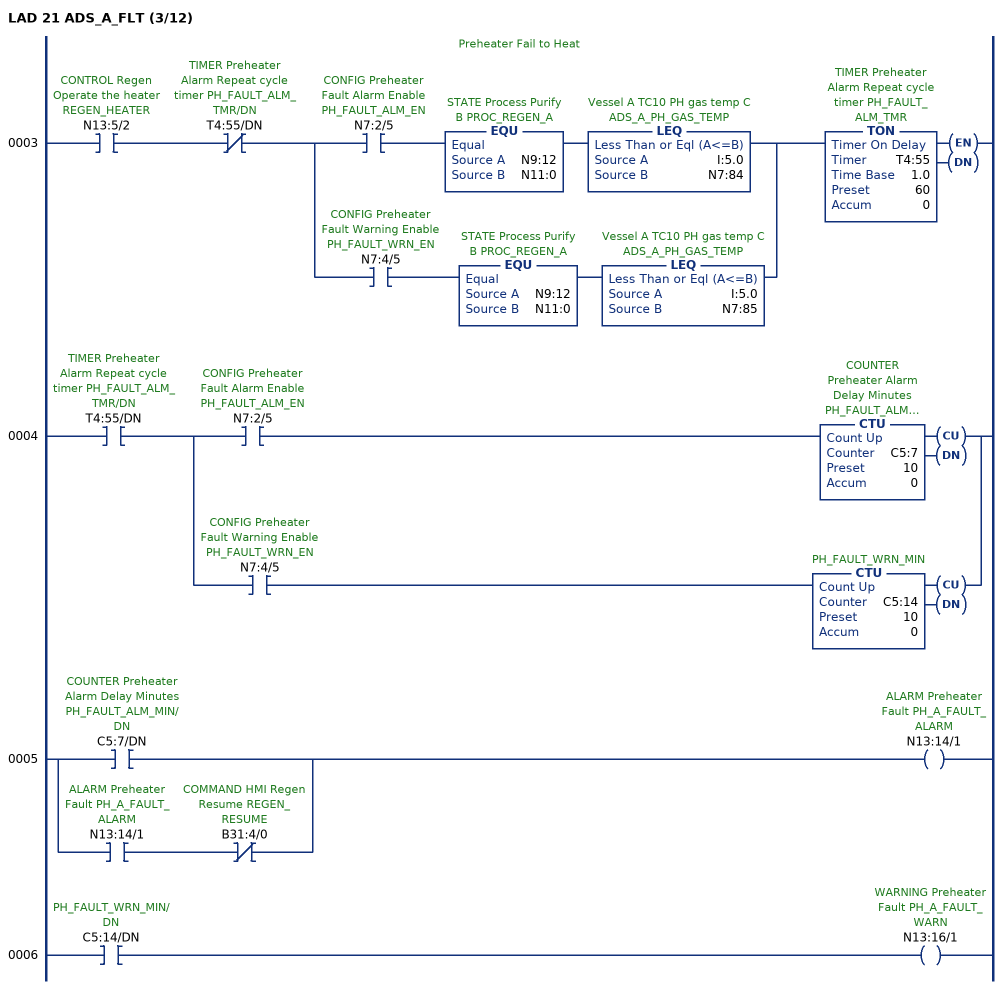
% Rung: 3 %
% Preheater Fail to Heat %
SOR XIC N13:5/2 XIO T4:55/DN BST XIC N7:2/5 EQU N9:12 N11:0 LEQ I:5.0 N7:84 NXB XIC N7:4/5 EQU N9:12 N11:0 LEQ I:5.0 N7:85 BND TON T4:55 1.0 60 0 EOR
%   N13:5/2  REGEN_HEATER  "CONTROL Regen Operate the heater" %
%   T4:55  PH_FAULT_ALM_TMR  "TIMER Preheater Alarm Repeat cycle timer" %
%   N7:2/5  PH_FAULT_ALM_EN  "CONFIG Preheater Fault Alarm Enable" %
%   N9:12  PROC_REGEN_A  "STATE Process Purify B" %
%   N11:0  PROC_STATE  "STATE The current state of the process" %
%   I:5.0  ADS_A_PH_GAS_TEMP  "Vessel A TC10 PH gas temp C" %
%   N7:84  PH_FAULT_ALARM_SP  "CONFIG Preheater Temperature Delta Alarm Setpoint" %
%   N7:4/5  PH_FAULT_WRN_EN  "CONFIG Preheater Fault Warning Enable" %
%   N7:85  PH_FAULT_WARN_SP %
% Rung: 4 %
SOR XIC T4:55/DN BST XIC N7:2/5 CTU C5:7 10 0 NXB XIC N7:4/5 CTU C5:14 10 0 BND EOR
%   T4:55  PH_FAULT_ALM_TMR  "TIMER Preheater Alarm Repeat cycle timer" %
%   N7:2/5  PH_FAULT_ALM_EN  "CONFIG Preheater Fault Alarm Enable" %
%   C5:7  PH_FAULT_ALM_MIN  "COUNTER Preheater Alarm Delay Minutes" %
%   N7:4/5  PH_FAULT_WRN_EN  "CONFIG Preheater Fault Warning Enable" %
%   C5:14  PH_FAULT_WRN_MIN %
% Rung: 5 %
SOR BST XIC C5:7/DN NXB XIC N13:14/1 XIO B31:4/0 BND OTE N13:14/1 EOR
%   C5:7  PH_FAULT_ALM_MIN  "COUNTER Preheater Alarm Delay Minutes" %
%   N13:14/1  PH_A_FAULT_ALARM  "ALARM Preheater Fault" %
%   B31:4/0  REGEN_RESUME  "COMMAND HMI Regen Resume" %
% Rung: 6 %
SOR XIC C5:14/DN OTE N13:16/1 EOR
%   C5:14  PH_FAULT_WRN_MIN %
%   N13:16/1  PH_A_FAULT_WARN  "WARNING Preheater Fault" %

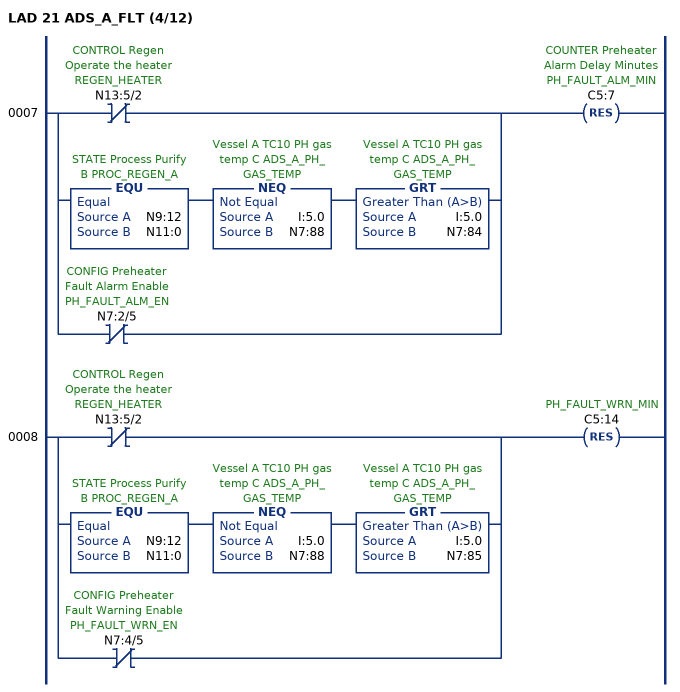
% Rung: 7 %
SOR BST XIO N13:5/2 NXB EQU N9:12 N11:0 NEQ I:5.0 N7:88 GRT I:5.0 N7:84 NXB XIO N7:2/5 BND RES C5:7 EOR
%   N13:5/2  REGEN_HEATER  "CONTROL Regen Operate the heater" %
%   N9:12  PROC_REGEN_A  "STATE Process Purify B" %
%   N11:0  PROC_STATE  "STATE The current state of the process" %
%   I:5.0  ADS_A_PH_GAS_TEMP  "Vessel A TC10 PH gas temp C" %
%   N7:88  TC_OPEN_SP  "CONFIG The value read by an open TC input" %
%   N7:84  PH_FAULT_ALARM_SP  "CONFIG Preheater Temperature Delta Alarm Setpoint" %
%   N7:2/5  PH_FAULT_ALM_EN  "CONFIG Preheater Fault Alarm Enable" %
%   C5:7  PH_FAULT_ALM_MIN  "COUNTER Preheater Alarm Delay Minutes" %
% Rung: 8 %
SOR BST XIO N13:5/2 NXB EQU N9:12 N11:0 NEQ I:5.0 N7:88 GRT I:5.0 N7:85 NXB XIO N7:4/5 BND RES C5:14 EOR
%   N13:5/2  REGEN_HEATER  "CONTROL Regen Operate the heater" %
%   N9:12  PROC_REGEN_A  "STATE Process Purify B" %
%   N11:0  PROC_STATE  "STATE The current state of the process" %
%   I:5.0  ADS_A_PH_GAS_TEMP  "Vessel A TC10 PH gas temp C" %
%   N7:88  TC_OPEN_SP  "CONFIG The value read by an open TC input" %
%   N7:85  PH_FAULT_WARN_SP %
%   N7:4/5  PH_FAULT_WRN_EN  "CONFIG Preheater Fault Warning Enable" %
%   C5:14  PH_FAULT_WRN_MIN %

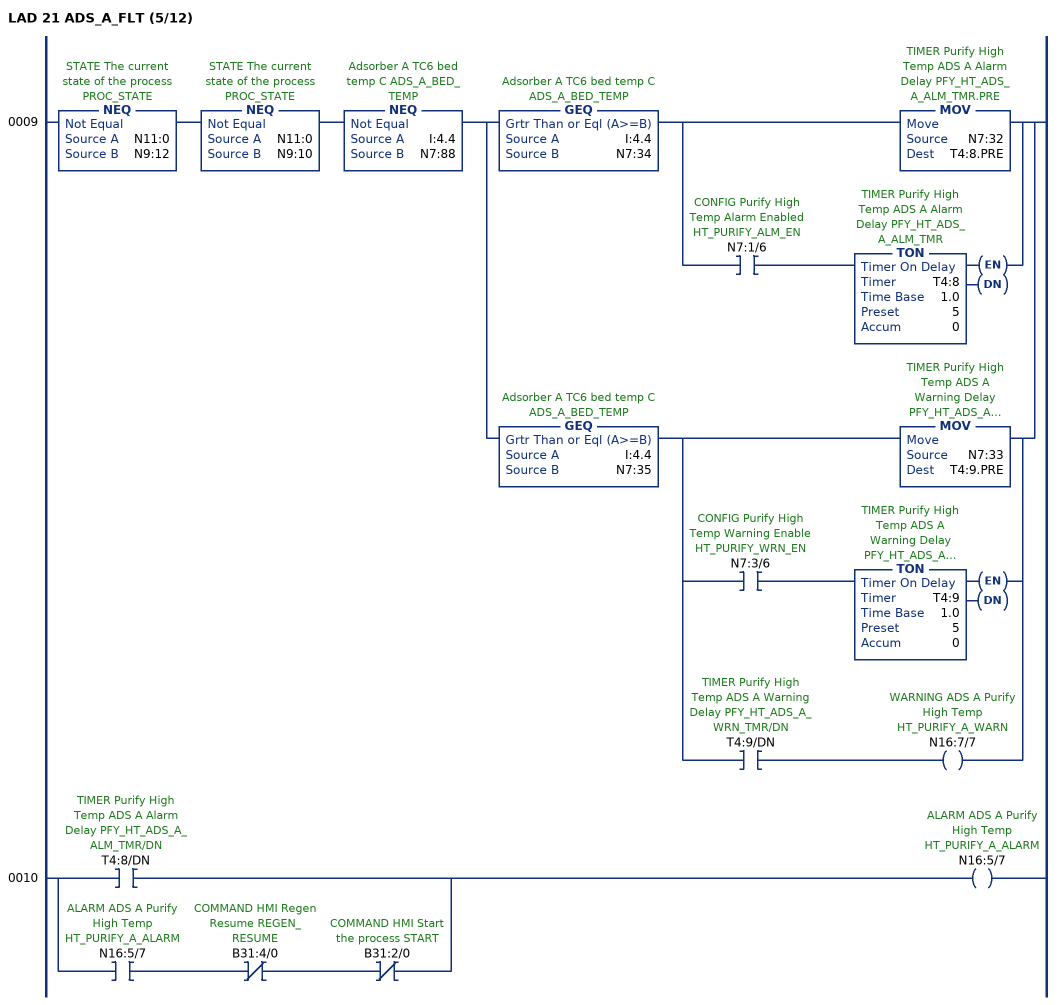
% Rung: 9 %
SOR NEQ N11:0 N9:12 NEQ N11:0 N9:10 NEQ I:4.4 N7:88 BST GEQ I:4.4 N7:34 BST MOV N7:32 T4:8.PRE NXB XIC N7:1/6 TON T4:8 1.0 5 0 BND NXB GEQ I:4.4 N7:35 BST MOV N7:33 T4:9.PRE NXB XIC N7:3/6 TON T4:9 1.0 5 0 NXB XIC T4:9/DN OTE N16:7/7 BND BND EOR
%   N11:0  PROC_STATE  "STATE The current state of the process" %
%   N9:12  PROC_REGEN_A  "STATE Process Purify B" %
%   N9:10  PROCESS_STANDBY %
%   I:4.4  ADS_A_BED_TEMP  "Adsorber A TC6 bed temp C" %
%   N7:88  TC_OPEN_SP  "CONFIG The value read by an open TC input" %
%   N7:34  HT_PURIFY_ALM_SP  "CONFIG Purify High Temp Alarm Setpoint" %
%   N7:32  HT_PURIFY_ALM_DLY  "CONFIG Purify High Temp Alarm Delay" %
%   T4:8  PFY_HT_ADS_A_ALM_TMR  "TIMER Purify High Temp ADS A Alarm Delay" %
%   N7:1/6  HT_PURIFY_ALM_EN  "CONFIG Purify High Temp Alarm Enabled" %
%   N7:35  HT_PURIFY_WRN_SP  "CONFIG Purify High Temp Warning Setpoint" %
%   N7:33  HT_PURIFY_WRN_DLY  "CONFIG Purify High Temp Warning Delay" %
%   T4:9  PFY_HT_ADS_A_WRN_TMR  "TIMER Purify High Temp ADS A Warning Delay" %
%   N7:3/6  HT_PURIFY_WRN_EN  "CONFIG Purify High Temp Warning Enable" %
%   N16:7/7  HT_PURIFY_A_WARN  "WARNING ADS A Purify High Temp" %
% Rung: 10 %
SOR BST XIC T4:8/DN NXB XIC N16:5/7 XIO B31:4/0 XIO B31:2/0 BND OTE N16:5/7 EOR
%   T4:8  PFY_HT_ADS_A_ALM_TMR  "TIMER Purify High Temp ADS A Alarm Delay" %
%   N16:5/7  HT_PURIFY_A_ALARM  "ALARM ADS A Purify High Temp" %
%   B31:4/0  REGEN_RESUME  "COMMAND HMI Regen Resume" %
%   B31:2/0  START  "COMMAND HMI Start the process" %

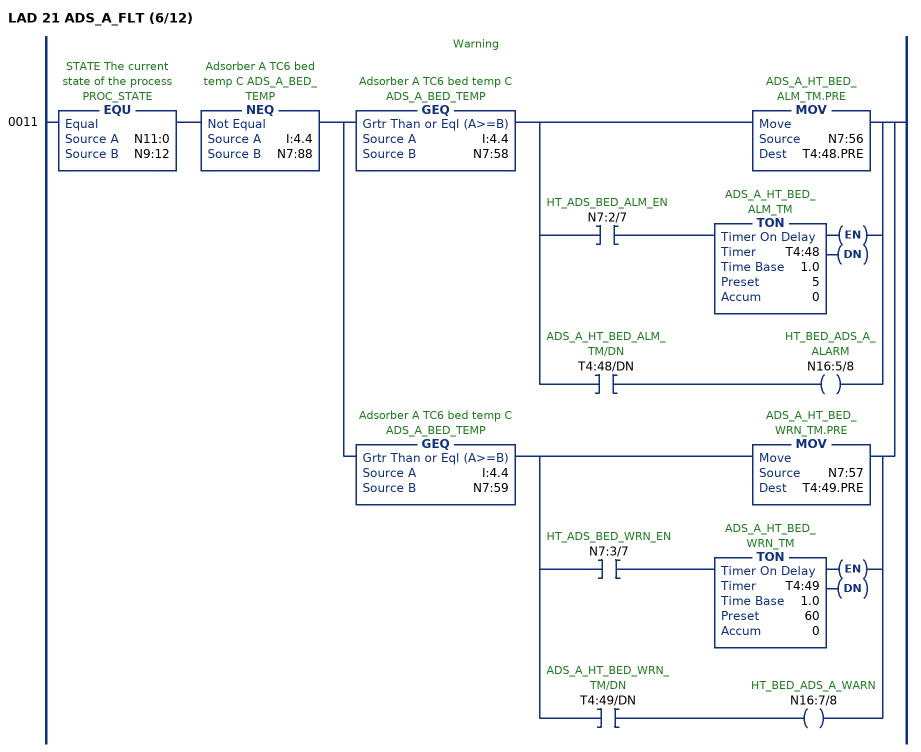
% Rung: 11 %
% Warning %
SOR EQU N11:0 N9:12 NEQ I:4.4 N7:88 BST GEQ I:4.4 N7:58 BST MOV N7:56 T4:48.PRE NXB XIC N7:2/7 TON T4:48 1.0 5 0 NXB XIC T4:48/DN OTE N16:5/8 BND NXB GEQ I:4.4 N7:59 BST MOV N7:57 T4:49.PRE NXB XIC N7:3/7 TON T4:49 1.0 60 0 NXB XIC T4:49/DN OTE N16:7/8 BND BND EOR
%   N11:0  PROC_STATE  "STATE The current state of the process" %
%   N9:12  PROC_REGEN_A  "STATE Process Purify B" %
%   I:4.4  ADS_A_BED_TEMP  "Adsorber A TC6 bed temp C" %
%   N7:88  TC_OPEN_SP  "CONFIG The value read by an open TC input" %
%   N7:58  HT_ADS_BED_ALM_SP %
%   N7:56  HT_ADS_BED_ALM_DLY %
%   T4:48  ADS_A_HT_BED_ALM_TM %
%   N7:2/7  HT_ADS_BED_ALM_EN %
%   N16:5/8  HT_BED_ADS_A_ALARM %
%   N7:59  HT_ADS_BED_WRN_SP %
%   N7:57  HT_ADS_BED_WRN_DLY %
%   T4:49  ADS_A_HT_BED_WRN_TM %
%   N7:3/7  HT_ADS_BED_WRN_EN %
%   N16:7/8  HT_BED_ADS_A_WARN %

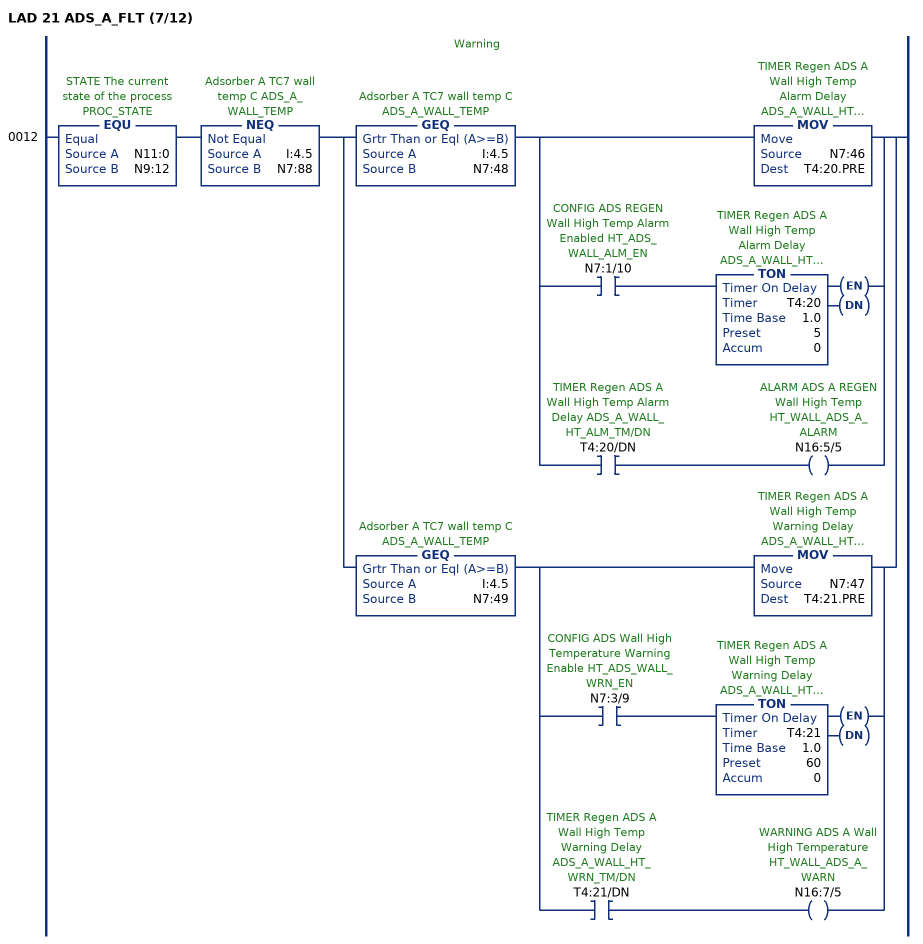
% Rung: 12 %
% Warning %
SOR EQU N11:0 N9:12 NEQ I:4.5 N7:88 BST GEQ I:4.5 N7:48 BST MOV N7:46 T4:20.PRE NXB XIC N7:1/10 TON T4:20 1.0 5 0 NXB XIC T4:20/DN OTE N16:5/5 BND NXB GEQ I:4.5 N7:49 BST MOV N7:47 T4:21.PRE NXB XIC N7:3/9 TON T4:21 1.0 60 0 NXB XIC T4:21/DN OTE N16:7/5 BND BND EOR
%   N11:0  PROC_STATE  "STATE The current state of the process" %
%   N9:12  PROC_REGEN_A  "STATE Process Purify B" %
%   I:4.5  ADS_A_WALL_TEMP  "Adsorber A TC7 wall temp C" %
%   N7:88  TC_OPEN_SP  "CONFIG The value read by an open TC input" %
%   N7:48  HT_ADS_WALL_ALM_SP  "CONFIG ADS Wall Regen High Temp Alarm" %
%   N7:46  HT_ADS_WALL_ALM_DLY  "CONFIG ADS Wall High Temperature Alarm Delay" %
%   T4:20  ADS_A_WALL_HT_ALM_TM  "TIMER Regen ADS A Wall High Temp Alarm Delay" %
%   N7:1/10  HT_ADS_WALL_ALM_EN  "CONFIG ADS REGEN Wall High Temp Alarm Enabled" %
%   N16:5/5  HT_WALL_ADS_A_ALARM  "ALARM ADS A REGEN Wall High Temp" %
%   N7:49  HT_ADS_WALL_WRN_SP  "CONFIG ADS Wall Regen High Temp Alarm" %
%   N7:47  HT_ADS_WALL_WRN_DLY  "CONFIG ADS Wall High Temperature Warning Delay" %
%   T4:21  ADS_A_WALL_HT_WRN_TM  "TIMER Regen ADS A Wall High Temp Warning Delay" %
%   N7:3/9  HT_ADS_WALL_WRN_EN  "CONFIG ADS Wall High Temperature Warning Enable" %
%   N16:7/5  HT_WALL_ADS_A_WARN  "WARNING ADS A Wall High Temperature" %

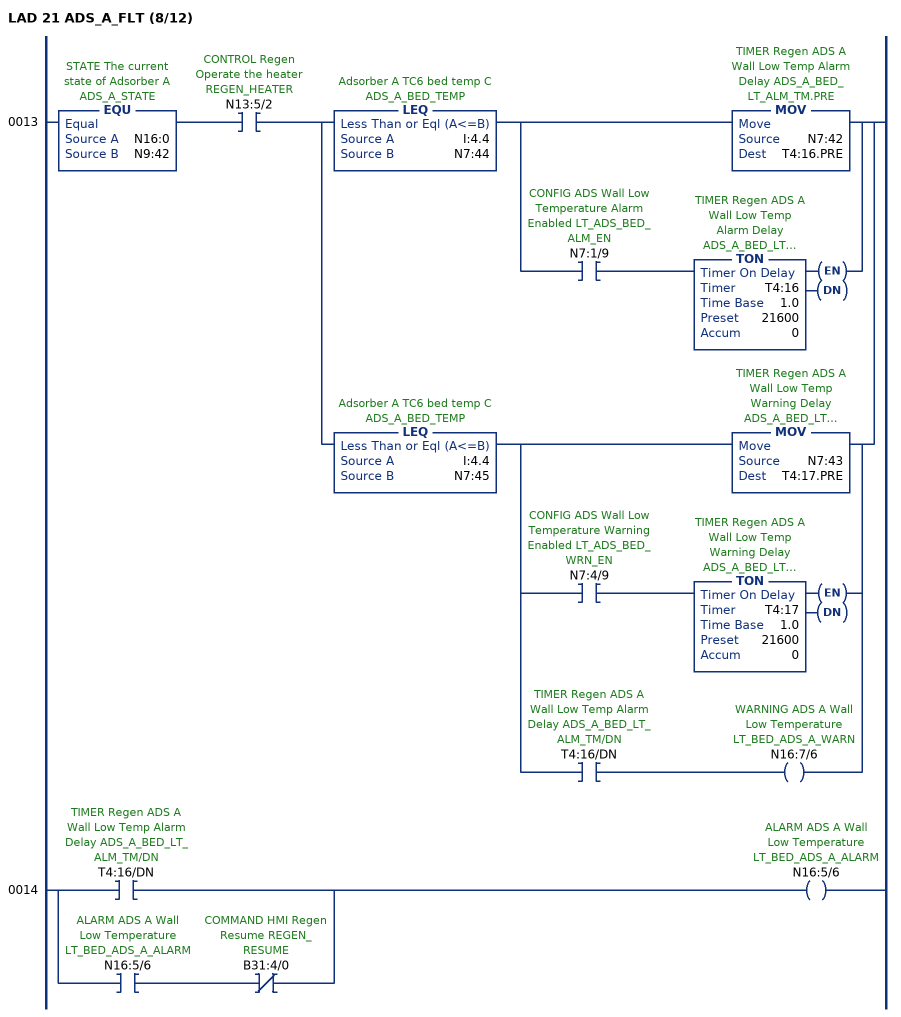
% Rung: 13 %
SOR EQU N16:0 N9:42 XIC N13:5/2 BST LEQ I:4.4 N7:44 BST MOV N7:42 T4:16.PRE NXB XIC N7:1/9 TON T4:16 1.0 21600 0 BND NXB LEQ I:4.4 N7:45 BST MOV N7:43 T4:17.PRE NXB XIC N7:4/9 TON T4:17 1.0 21600 0 NXB XIC T4:16/DN OTE N16:7/6 BND BND EOR
%   N16:0  ADS_A_STATE  "STATE The current state of Adsorber A" %
%   N9:42  ADS_REGEN  "STATE ADS Regen" %
%   N13:5/2  REGEN_HEATER  "CONTROL Regen Operate the heater" %
%   I:4.4  ADS_A_BED_TEMP  "Adsorber A TC6 bed temp C" %
%   N7:44  LT_ADS_BED_ALM_SP  "CONFIG ADS Wall Regen Heat Low Temperature Alarm Setpoint" %
%   N7:42  LT_ADS_BED_ALM_DLY  "CONFIG ADS Wall Regen heat Low Temperature Alarm Delay" %
%   T4:16  ADS_A_BED_LT_ALM_TM  "TIMER Regen ADS A Wall Low Temp Alarm Delay" %
%   N7:1/9  LT_ADS_BED_ALM_EN  "CONFIG ADS Wall Low Temperature Alarm Enabled" %
%   N7:45  LT_ADS_BED_WRN_SP  "CONFIG ADS Wall Regen Heat Low Temperature Warning Setpoint" %
%   N7:43  LT_ADS_BED_WRN_DLY  "CONFIG ADS Wall Regen heat Low Temperature Warning Delay" %
%   T4:17  ADS_A_BED_LT_WRN_TM  "TIMER Regen ADS A Wall Low Temp Warning Delay" %
%   N7:4/9  LT_ADS_BED_WRN_EN  "CONFIG ADS Wall Low Temperature Warning Enabled" %
%   N16:7/6  LT_BED_ADS_A_WARN  "WARNING ADS A Wall Low Temperature" %
% Rung: 14 %
SOR BST XIC T4:16/DN NXB XIC N16:5/6 XIO B31:4/0 BND OTE N16:5/6 EOR
%   T4:16  ADS_A_BED_LT_ALM_TM  "TIMER Regen ADS A Wall Low Temp Alarm Delay" %
%   N16:5/6  LT_BED_ADS_A_ALARM  "ALARM ADS A Wall Low Temperature" %
%   B31:4/0  REGEN_RESUME  "COMMAND HMI Regen Resume" %

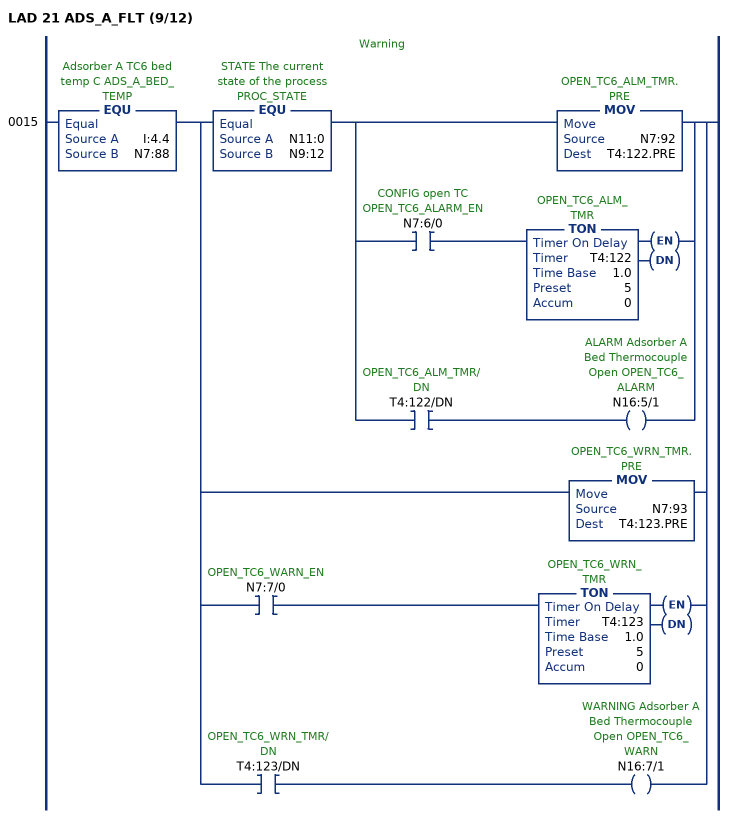
% Rung: 15 %
% Warning %
SOR EQU I:4.4 N7:88 BST EQU N11:0 N9:12 BST MOV N7:92 T4:122.PRE NXB XIC N7:6/0 TON T4:122 1.0 5 0 NXB XIC T4:122/DN OTE N16:5/1 BND NXB MOV N7:93 T4:123.PRE NXB XIC N7:7/0 TON T4:123 1.0 5 0 NXB XIC T4:123/DN OTE N16:7/1 BND EOR
%   I:4.4  ADS_A_BED_TEMP  "Adsorber A TC6 bed temp C" %
%   N7:88  TC_OPEN_SP  "CONFIG The value read by an open TC input" %
%   N11:0  PROC_STATE  "STATE The current state of the process" %
%   N9:12  PROC_REGEN_A  "STATE Process Purify B" %
%   N7:92  OPEN_TC_ALM_DLY %
%   T4:122  OPEN_TC6_ALM_TMR %
%   N7:6/0  OPEN_TC6_ALARM_EN  "CONFIG open TC" %
%   N16:5/1  OPEN_TC6_ALARM  "ALARM Adsorber A Bed Thermocouple Open" %
%   N7:93  OPEN_TC_WRN_DLY %
%   T4:123  OPEN_TC6_WRN_TMR %
%   N7:7/0  OPEN_TC6_WARN_EN %
%   N16:7/1  OPEN_TC6_WARN  "WARNING Adsorber A Bed Thermocouple Open" %

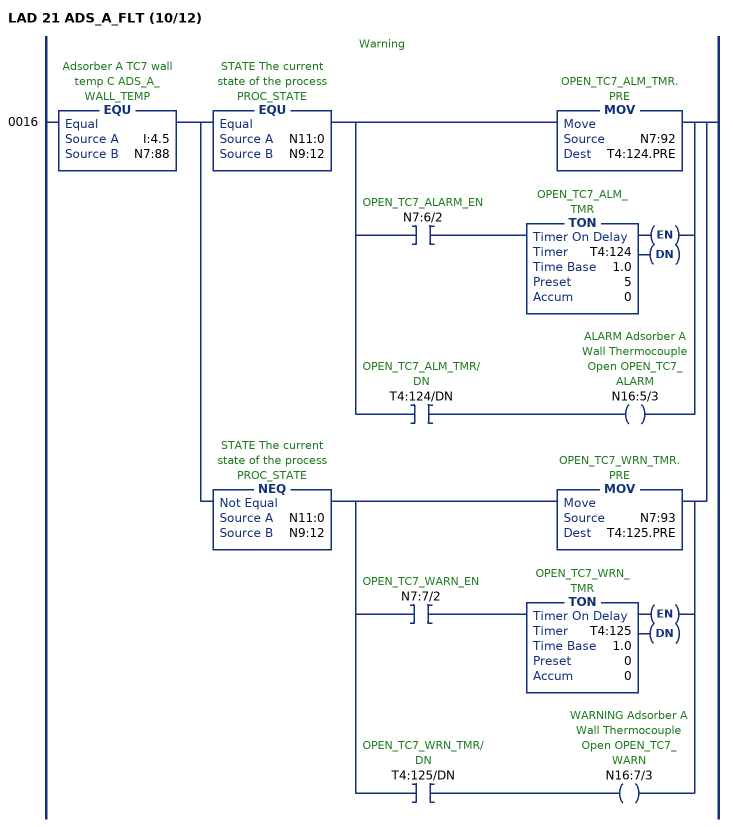
% Rung: 16 %
% Warning %
SOR EQU I:4.5 N7:88 BST EQU N11:0 N9:12 BST MOV N7:92 T4:124.PRE NXB XIC N7:6/2 TON T4:124 1.0 5 0 NXB XIC T4:124/DN OTE N16:5/3 BND NXB NEQ N11:0 N9:12 BST MOV N7:93 T4:125.PRE NXB XIC N7:7/2 TON T4:125 1.0 0 0 NXB XIC T4:125/DN OTE N16:7/3 BND BND EOR
%   I:4.5  ADS_A_WALL_TEMP  "Adsorber A TC7 wall temp C" %
%   N7:88  TC_OPEN_SP  "CONFIG The value read by an open TC input" %
%   N11:0  PROC_STATE  "STATE The current state of the process" %
%   N9:12  PROC_REGEN_A  "STATE Process Purify B" %
%   N7:92  OPEN_TC_ALM_DLY %
%   T4:124  OPEN_TC7_ALM_TMR %
%   N7:6/2  OPEN_TC7_ALARM_EN %
%   N16:5/3  OPEN_TC7_ALARM  "ALARM Adsorber A Wall Thermocouple Open" %
%   N7:93  OPEN_TC_WRN_DLY %
%   T4:125  OPEN_TC7_WRN_TMR %
%   N7:7/2  OPEN_TC7_WARN_EN %
%   N16:7/3  OPEN_TC7_WARN  "WARNING Adsorber A Wall Thermocouple Open" %

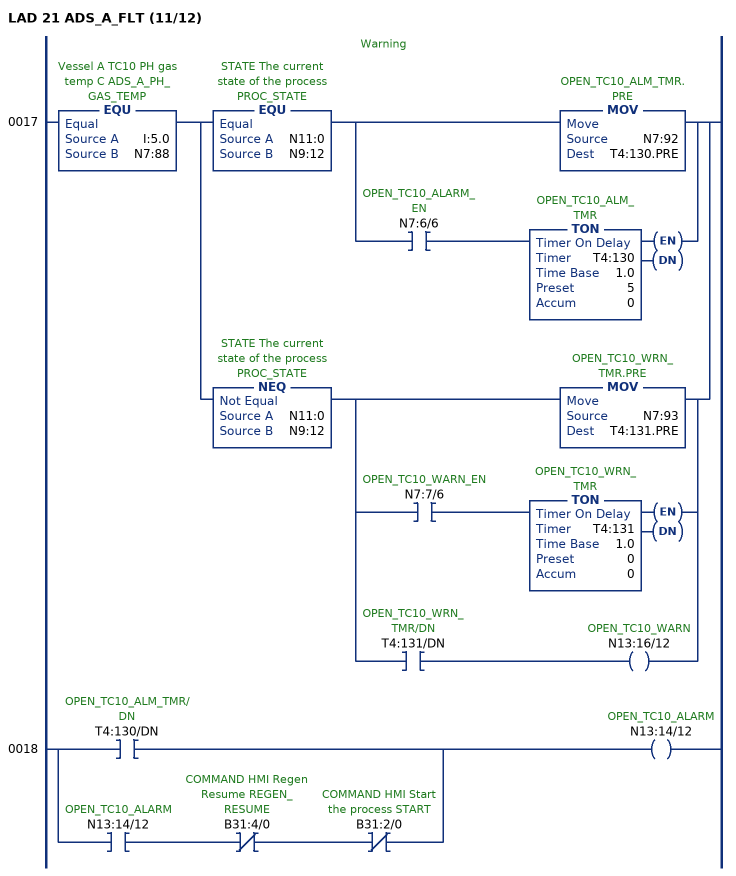
% Rung: 17 %
% Warning %
SOR EQU I:5.0 N7:88 BST EQU N11:0 N9:12 BST MOV N7:92 T4:130.PRE NXB XIC N7:6/6 TON T4:130 1.0 5 0 BND NXB NEQ N11:0 N9:12 BST MOV N7:93 T4:131.PRE NXB XIC N7:7/6 TON T4:131 1.0 0 0 NXB XIC T4:131/DN OTE N13:16/12 BND BND EOR
%   I:5.0  ADS_A_PH_GAS_TEMP  "Vessel A TC10 PH gas temp C" %
%   N7:88  TC_OPEN_SP  "CONFIG The value read by an open TC input" %
%   N11:0  PROC_STATE  "STATE The current state of the process" %
%   N9:12  PROC_REGEN_A  "STATE Process Purify B" %
%   N7:92  OPEN_TC_ALM_DLY %
%   T4:130  OPEN_TC10_ALM_TMR %
%   N7:6/6  OPEN_TC10_ALARM_EN %
%   N7:93  OPEN_TC_WRN_DLY %
%   T4:131  OPEN_TC10_WRN_TMR %
%   N7:7/6  OPEN_TC10_WARN_EN %
%   N13:16/12  OPEN_TC10_WARN %
% Rung: 18 %
SOR BST XIC T4:130/DN NXB XIC N13:14/12 XIO B31:4/0 XIO B31:2/0 BND OTE N13:14/12 EOR
%   T4:130  OPEN_TC10_ALM_TMR %
%   N13:14/12  OPEN_TC10_ALARM %
%   B31:4/0  REGEN_RESUME  "COMMAND HMI Regen Resume" %
%   B31:2/0  START  "COMMAND HMI Start the process" %

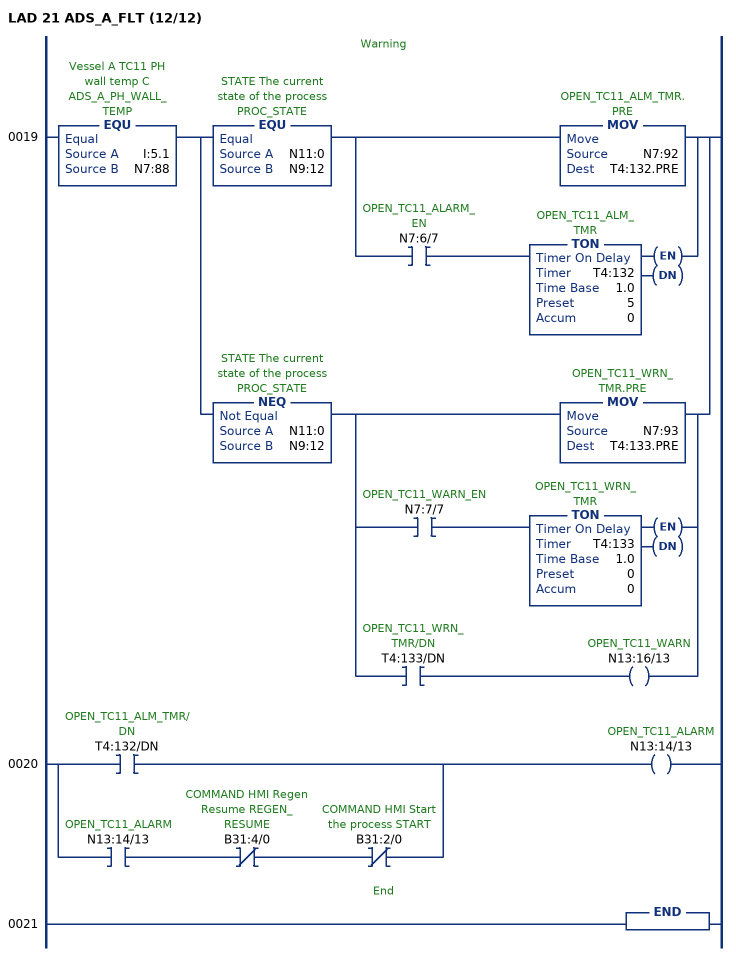
% Rung: 19 %
% Warning %
SOR EQU I:5.1 N7:88 BST EQU N11:0 N9:12 BST MOV N7:92 T4:132.PRE NXB XIC N7:6/7 TON T4:132 1.0 5 0 BND NXB NEQ N11:0 N9:12 BST MOV N7:93 T4:133.PRE NXB XIC N7:7/7 TON T4:133 1.0 0 0 NXB XIC T4:133/DN OTE N13:16/13 BND BND EOR
%   I:5.1  ADS_A_PH_WALL_TEMP  "Vessel A TC11 PH wall temp C" %
%   N7:88  TC_OPEN_SP  "CONFIG The value read by an open TC input" %
%   N11:0  PROC_STATE  "STATE The current state of the process" %
%   N9:12  PROC_REGEN_A  "STATE Process Purify B" %
%   N7:92  OPEN_TC_ALM_DLY %
%   T4:132  OPEN_TC11_ALM_TMR %
%   N7:6/7  OPEN_TC11_ALARM_EN %
%   N7:93  OPEN_TC_WRN_DLY %
%   T4:133  OPEN_TC11_WRN_TMR %
%   N7:7/7  OPEN_TC11_WARN_EN %
%   N13:16/13  OPEN_TC11_WARN %
% Rung: 20 %
SOR BST XIC T4:132/DN NXB XIC N13:14/13 XIO B31:4/0 XIO B31:2/0 BND OTE N13:14/13 EOR
%   T4:132  OPEN_TC11_ALM_TMR %
%   N13:14/13  OPEN_TC11_ALARM %
%   B31:4/0  REGEN_RESUME  "COMMAND HMI Regen Resume" %
%   B31:2/0  START  "COMMAND HMI Start the process" %
% Rung: 21 %
% End %
SOR END EOR

LADDER 22 "ADS_B"    % Controld Adsorber B %
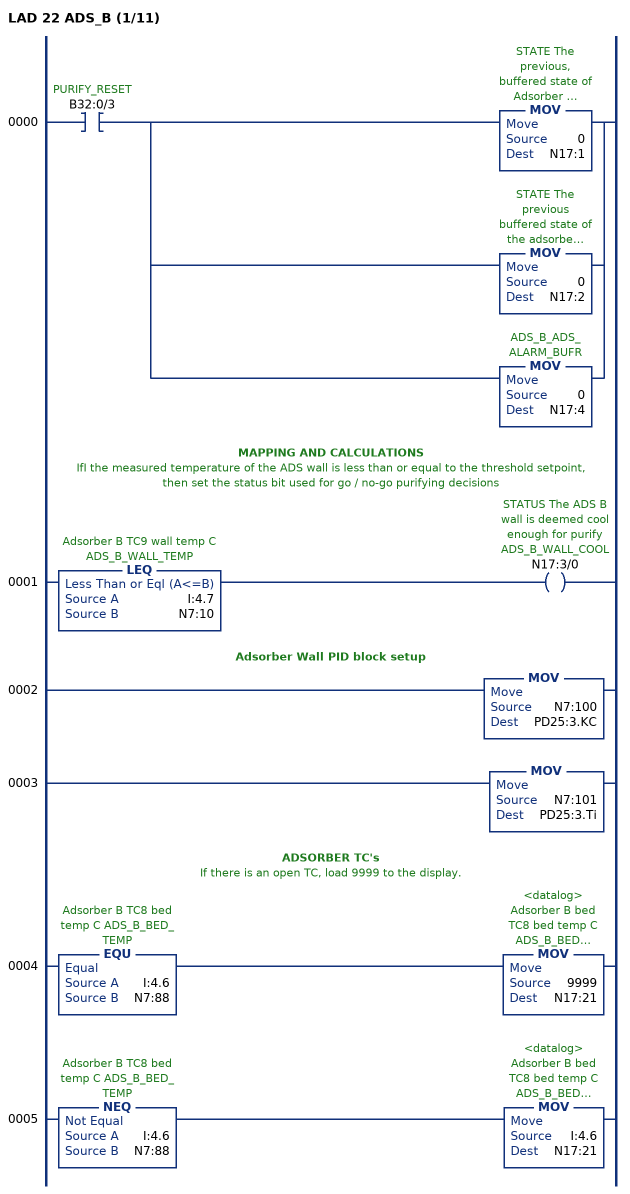
% Rung: 0 %
SOR XIC B32:0/3 BST MOV 0 N17:1 NXB MOV 0 N17:2 NXB MOV 0 N17:4 BND EOR
%   B32:0/3  PURIFY_RESET %
%   N17:1  ADS_B_STANDBY_BUFFER  "STATE The previous, buffered state of Adsorber B" %
%   N17:2  ADS_B_SYS_ALARM_BUFR  "STATE The previous buffered state of the adsorber when the alarm occured" %
%   N17:4  ADS_B_ADS_ALARM_BUFR %
% Rung: 1 %
% TITLE: MAPPING AND CALCULATIONS %
% IfI the measured temperature of the ADS wall is less than or equal to the threshold setpoint, then set the status bit used for go / no-go purifying decisions %
SOR LEQ I:4.7 N7:10 OTE N17:3/0 EOR
%   I:4.7  ADS_B_WALL_TEMP  "Adsorber B TC9 wall temp C" %
%   N7:10  ADS_WALL_TEMP_COOL  "CONFIG The temp at which the adsorber wall is deemed to be cool enough to purify" %
%   N17:3/0  ADS_B_WALL_COOL  "STATUS The ADS B wall is deemed cool enough for purify" %
% Rung: 2 %
% TITLE: Adsorber Wall PID block setup %
SOR MOV N7:100 PD25:3.KC EOR
%   N7:100  BLANKET_P  "CONFIG Blanket Proportional Gain New" %
% Rung: 3 %
SOR MOV N7:101 PD25:3.Ti EOR
%   N7:101  BLANKET_I  "CONFIG Blanket Integral Gain New" %
% Rung: 4 %
% TITLE: ADSORBER TC's %
% If there is an open TC, load 9999 to the display. %
SOR EQU I:4.6 N7:88 MOV 9999 N17:21 EOR
%   I:4.6  ADS_B_BED_TEMP  "Adsorber B TC8 bed temp C" %
%   N7:88  TC_OPEN_SP  "CONFIG The value read by an open TC input" %
%   N17:21  ADS_B_BED_TEMP_READ  "<datalog> Adsorber B bed TC8 bed temp C" %
% Rung: 5 %
SOR NEQ I:4.6 N7:88 MOV I:4.6 N17:21 EOR
%   I:4.6  ADS_B_BED_TEMP  "Adsorber B TC8 bed temp C" %
%   N7:88  TC_OPEN_SP  "CONFIG The value read by an open TC input" %
%   N17:21  ADS_B_BED_TEMP_READ  "<datalog> Adsorber B bed TC8 bed temp C" %

